// TIA Portal V18 export
FUNCTION "SS2_A4_32DO_IO_Update" : Void   // FC11150, LAD
{ S7_Optimized_Access := 'TRUE' }
VERSION : 0.1
// stored: AutoNumber false, IsIECCheckEnabled false, SetENOAutomatically false, UDAEnableTagReadback false
BEGIN

REGION Network 1: DQa0
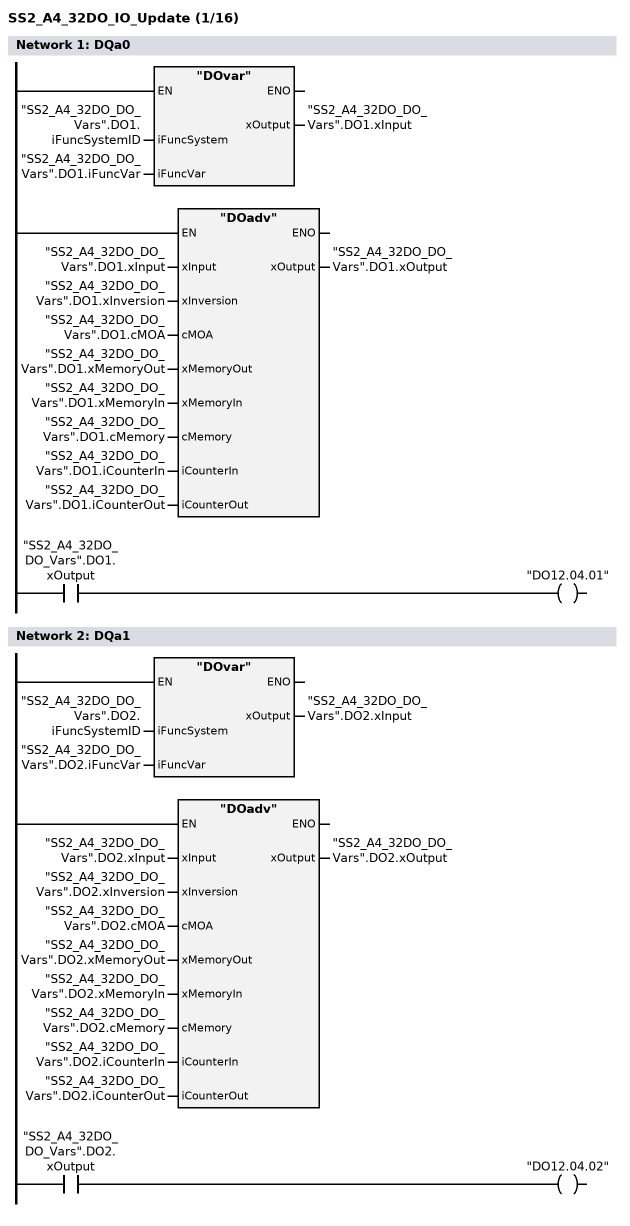
   RUNG wire#powerrail
      "DOvar"(iFuncSystem := "SS2_A4_32DO_DO_Vars".DO1.iFuncSystemID, iFuncVar := "SS2_A4_32DO_DO_Vars".DO1.iFuncVar, xOutput => "SS2_A4_32DO_DO_Vars".DO1.xInput)
   END_RUNG
   RUNG wire#powerrail
      "DOadv"(xInput := "SS2_A4_32DO_DO_Vars".DO1.xInput, xInversion := "SS2_A4_32DO_DO_Vars".DO1.xInversion, cMOA := "SS2_A4_32DO_DO_Vars".DO1.cMOA, xMemoryOut := "SS2_A4_32DO_DO_Vars".DO1.xMemoryOut, xMemoryIn := "SS2_A4_32DO_DO_Vars".DO1.xMemoryIn, cMemory := "SS2_A4_32DO_DO_Vars".DO1.cMemory, iCounterIn := "SS2_A4_32DO_DO_Vars".DO1.iCounterIn, iCounterOut := "SS2_A4_32DO_DO_Vars".DO1.iCounterOut, xOutput => "SS2_A4_32DO_DO_Vars".DO1.xOutput)
   END_RUNG
   RUNG wire#powerrail
      Contact( "SS2_A4_32DO_DO_Vars".DO1.xOutput )
      Coil( "DO12.04.01" )
   END_RUNG
   // the same network as SCL:
   "DOvar"(iFuncSystem := "SS2_A4_32DO_DO_Vars".DO1.iFuncSystemID,
           iFuncVar := "SS2_A4_32DO_DO_Vars".DO1.iFuncVar,
           xOutput => "SS2_A4_32DO_DO_Vars".DO1.xInput);
   "DOadv"(xInput := "SS2_A4_32DO_DO_Vars".DO1.xInput,
           xInversion := "SS2_A4_32DO_DO_Vars".DO1.xInversion,
           cMOA := "SS2_A4_32DO_DO_Vars".DO1.cMOA,
           xMemoryOut := "SS2_A4_32DO_DO_Vars".DO1.xMemoryOut,
           xMemoryIn := "SS2_A4_32DO_DO_Vars".DO1.xMemoryIn,
           cMemory := "SS2_A4_32DO_DO_Vars".DO1.cMemory,
           iCounterIn := "SS2_A4_32DO_DO_Vars".DO1.iCounterIn,
           iCounterOut := "SS2_A4_32DO_DO_Vars".DO1.iCounterOut,
           xOutput => "SS2_A4_32DO_DO_Vars".DO1.xOutput);
   "DO12.04.01" := "SS2_A4_32DO_DO_Vars".DO1.xOutput;
END_REGION

REGION Network 2: DQa1
   RUNG wire#powerrail
      "DOvar"(iFuncSystem := "SS2_A4_32DO_DO_Vars".DO2.iFuncSystemID, iFuncVar := "SS2_A4_32DO_DO_Vars".DO2.iFuncVar, xOutput => "SS2_A4_32DO_DO_Vars".DO2.xInput)
   END_RUNG
   RUNG wire#powerrail
      "DOadv"(xInput := "SS2_A4_32DO_DO_Vars".DO2.xInput, xInversion := "SS2_A4_32DO_DO_Vars".DO2.xInversion, cMOA := "SS2_A4_32DO_DO_Vars".DO2.cMOA, xMemoryOut := "SS2_A4_32DO_DO_Vars".DO2.xMemoryOut, xMemoryIn := "SS2_A4_32DO_DO_Vars".DO2.xMemoryIn, cMemory := "SS2_A4_32DO_DO_Vars".DO2.cMemory, iCounterIn := "SS2_A4_32DO_DO_Vars".DO2.iCounterIn, iCounterOut := "SS2_A4_32DO_DO_Vars".DO2.iCounterOut, xOutput => "SS2_A4_32DO_DO_Vars".DO2.xOutput)
   END_RUNG
   RUNG wire#powerrail
      Contact( "SS2_A4_32DO_DO_Vars".DO2.xOutput )
      Coil( "DO12.04.02" )
   END_RUNG
   // the same network as SCL:
   "DOvar"(iFuncSystem := "SS2_A4_32DO_DO_Vars".DO2.iFuncSystemID,
           iFuncVar := "SS2_A4_32DO_DO_Vars".DO2.iFuncVar,
           xOutput => "SS2_A4_32DO_DO_Vars".DO2.xInput);
   "DOadv"(xInput := "SS2_A4_32DO_DO_Vars".DO2.xInput,
           xInversion := "SS2_A4_32DO_DO_Vars".DO2.xInversion,
           cMOA := "SS2_A4_32DO_DO_Vars".DO2.cMOA,
           xMemoryOut := "SS2_A4_32DO_DO_Vars".DO2.xMemoryOut,
           xMemoryIn := "SS2_A4_32DO_DO_Vars".DO2.xMemoryIn,
           cMemory := "SS2_A4_32DO_DO_Vars".DO2.cMemory,
           iCounterIn := "SS2_A4_32DO_DO_Vars".DO2.iCounterIn,
           iCounterOut := "SS2_A4_32DO_DO_Vars".DO2.iCounterOut,
           xOutput => "SS2_A4_32DO_DO_Vars".DO2.xOutput);
   "DO12.04.02" := "SS2_A4_32DO_DO_Vars".DO2.xOutput;
END_REGION

REGION Network 3: DQa2
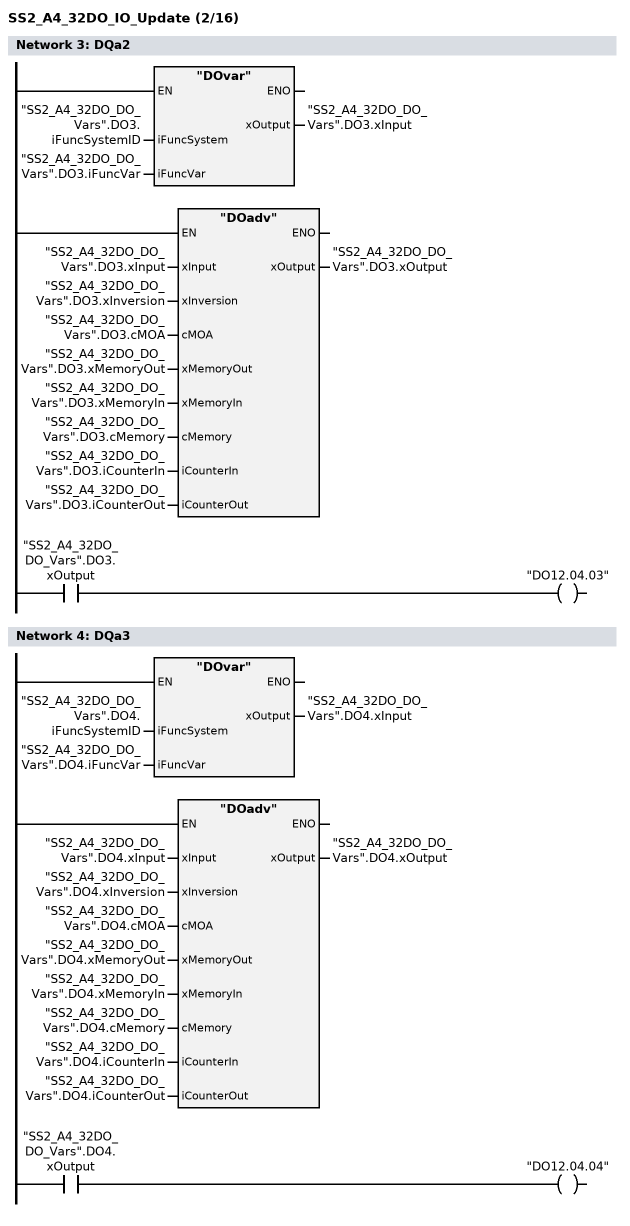
   RUNG wire#powerrail
      "DOvar"(iFuncSystem := "SS2_A4_32DO_DO_Vars".DO3.iFuncSystemID, iFuncVar := "SS2_A4_32DO_DO_Vars".DO3.iFuncVar, xOutput => "SS2_A4_32DO_DO_Vars".DO3.xInput)
   END_RUNG
   RUNG wire#powerrail
      "DOadv"(xInput := "SS2_A4_32DO_DO_Vars".DO3.xInput, xInversion := "SS2_A4_32DO_DO_Vars".DO3.xInversion, cMOA := "SS2_A4_32DO_DO_Vars".DO3.cMOA, xMemoryOut := "SS2_A4_32DO_DO_Vars".DO3.xMemoryOut, xMemoryIn := "SS2_A4_32DO_DO_Vars".DO3.xMemoryIn, cMemory := "SS2_A4_32DO_DO_Vars".DO3.cMemory, iCounterIn := "SS2_A4_32DO_DO_Vars".DO3.iCounterIn, iCounterOut := "SS2_A4_32DO_DO_Vars".DO3.iCounterOut, xOutput => "SS2_A4_32DO_DO_Vars".DO3.xOutput)
   END_RUNG
   RUNG wire#powerrail
      Contact( "SS2_A4_32DO_DO_Vars".DO3.xOutput )
      Coil( "DO12.04.03" )
   END_RUNG
   // the same network as SCL:
   "DOvar"(iFuncSystem := "SS2_A4_32DO_DO_Vars".DO3.iFuncSystemID,
           iFuncVar := "SS2_A4_32DO_DO_Vars".DO3.iFuncVar,
           xOutput => "SS2_A4_32DO_DO_Vars".DO3.xInput);
   "DOadv"(xInput := "SS2_A4_32DO_DO_Vars".DO3.xInput,
           xInversion := "SS2_A4_32DO_DO_Vars".DO3.xInversion,
           cMOA := "SS2_A4_32DO_DO_Vars".DO3.cMOA,
           xMemoryOut := "SS2_A4_32DO_DO_Vars".DO3.xMemoryOut,
           xMemoryIn := "SS2_A4_32DO_DO_Vars".DO3.xMemoryIn,
           cMemory := "SS2_A4_32DO_DO_Vars".DO3.cMemory,
           iCounterIn := "SS2_A4_32DO_DO_Vars".DO3.iCounterIn,
           iCounterOut := "SS2_A4_32DO_DO_Vars".DO3.iCounterOut,
           xOutput => "SS2_A4_32DO_DO_Vars".DO3.xOutput);
   "DO12.04.03" := "SS2_A4_32DO_DO_Vars".DO3.xOutput;
END_REGION

REGION Network 4: DQa3
   RUNG wire#powerrail
      "DOvar"(iFuncSystem := "SS2_A4_32DO_DO_Vars".DO4.iFuncSystemID, iFuncVar := "SS2_A4_32DO_DO_Vars".DO4.iFuncVar, xOutput => "SS2_A4_32DO_DO_Vars".DO4.xInput)
   END_RUNG
   RUNG wire#powerrail
      "DOadv"(xInput := "SS2_A4_32DO_DO_Vars".DO4.xInput, xInversion := "SS2_A4_32DO_DO_Vars".DO4.xInversion, cMOA := "SS2_A4_32DO_DO_Vars".DO4.cMOA, xMemoryOut := "SS2_A4_32DO_DO_Vars".DO4.xMemoryOut, xMemoryIn := "SS2_A4_32DO_DO_Vars".DO4.xMemoryIn, cMemory := "SS2_A4_32DO_DO_Vars".DO4.cMemory, iCounterIn := "SS2_A4_32DO_DO_Vars".DO4.iCounterIn, iCounterOut := "SS2_A4_32DO_DO_Vars".DO4.iCounterOut, xOutput => "SS2_A4_32DO_DO_Vars".DO4.xOutput)
   END_RUNG
   RUNG wire#powerrail
      Contact( "SS2_A4_32DO_DO_Vars".DO4.xOutput )
      Coil( "DO12.04.04" )
   END_RUNG
   // the same network as SCL:
   "DOvar"(iFuncSystem := "SS2_A4_32DO_DO_Vars".DO4.iFuncSystemID,
           iFuncVar := "SS2_A4_32DO_DO_Vars".DO4.iFuncVar,
           xOutput => "SS2_A4_32DO_DO_Vars".DO4.xInput);
   "DOadv"(xInput := "SS2_A4_32DO_DO_Vars".DO4.xInput,
           xInversion := "SS2_A4_32DO_DO_Vars".DO4.xInversion,
           cMOA := "SS2_A4_32DO_DO_Vars".DO4.cMOA,
           xMemoryOut := "SS2_A4_32DO_DO_Vars".DO4.xMemoryOut,
           xMemoryIn := "SS2_A4_32DO_DO_Vars".DO4.xMemoryIn,
           cMemory := "SS2_A4_32DO_DO_Vars".DO4.cMemory,
           iCounterIn := "SS2_A4_32DO_DO_Vars".DO4.iCounterIn,
           iCounterOut := "SS2_A4_32DO_DO_Vars".DO4.iCounterOut,
           xOutput => "SS2_A4_32DO_DO_Vars".DO4.xOutput);
   "DO12.04.04" := "SS2_A4_32DO_DO_Vars".DO4.xOutput;
END_REGION

REGION Network 5: DQa4
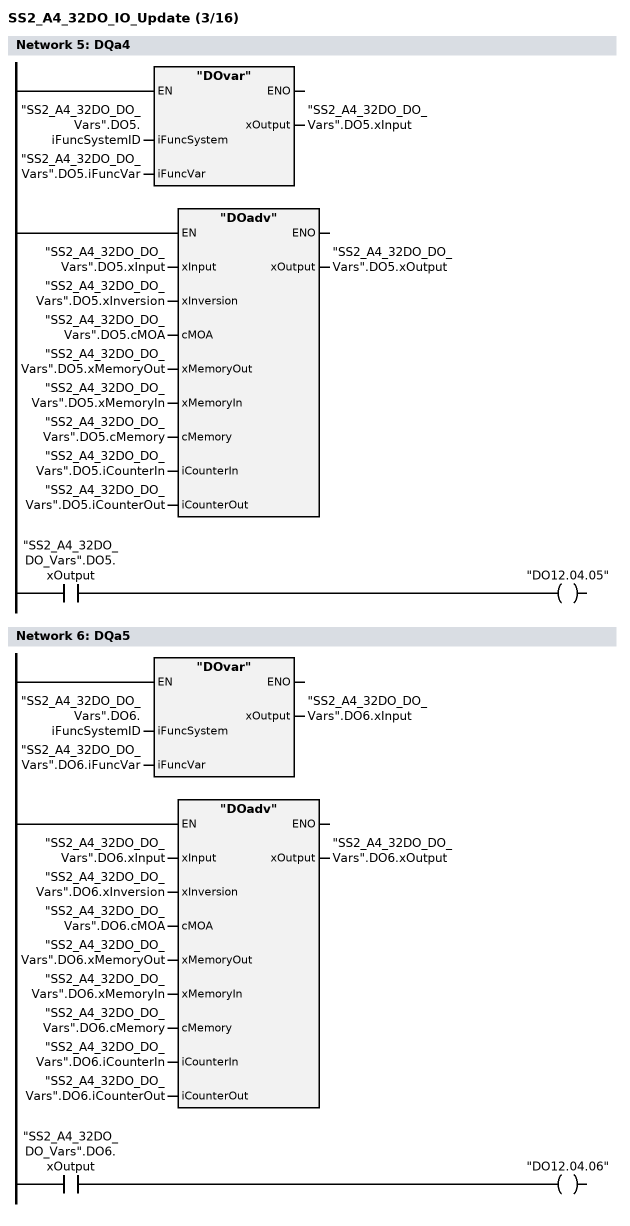
   RUNG wire#powerrail
      "DOvar"(iFuncSystem := "SS2_A4_32DO_DO_Vars".DO5.iFuncSystemID, iFuncVar := "SS2_A4_32DO_DO_Vars".DO5.iFuncVar, xOutput => "SS2_A4_32DO_DO_Vars".DO5.xInput)
   END_RUNG
   RUNG wire#powerrail
      "DOadv"(xInput := "SS2_A4_32DO_DO_Vars".DO5.xInput, xInversion := "SS2_A4_32DO_DO_Vars".DO5.xInversion, cMOA := "SS2_A4_32DO_DO_Vars".DO5.cMOA, xMemoryOut := "SS2_A4_32DO_DO_Vars".DO5.xMemoryOut, xMemoryIn := "SS2_A4_32DO_DO_Vars".DO5.xMemoryIn, cMemory := "SS2_A4_32DO_DO_Vars".DO5.cMemory, iCounterIn := "SS2_A4_32DO_DO_Vars".DO5.iCounterIn, iCounterOut := "SS2_A4_32DO_DO_Vars".DO5.iCounterOut, xOutput => "SS2_A4_32DO_DO_Vars".DO5.xOutput)
   END_RUNG
   RUNG wire#powerrail
      Contact( "SS2_A4_32DO_DO_Vars".DO5.xOutput )
      Coil( "DO12.04.05" )
   END_RUNG
   // the same network as SCL:
   "DOvar"(iFuncSystem := "SS2_A4_32DO_DO_Vars".DO5.iFuncSystemID,
           iFuncVar := "SS2_A4_32DO_DO_Vars".DO5.iFuncVar,
           xOutput => "SS2_A4_32DO_DO_Vars".DO5.xInput);
   "DOadv"(xInput := "SS2_A4_32DO_DO_Vars".DO5.xInput,
           xInversion := "SS2_A4_32DO_DO_Vars".DO5.xInversion,
           cMOA := "SS2_A4_32DO_DO_Vars".DO5.cMOA,
           xMemoryOut := "SS2_A4_32DO_DO_Vars".DO5.xMemoryOut,
           xMemoryIn := "SS2_A4_32DO_DO_Vars".DO5.xMemoryIn,
           cMemory := "SS2_A4_32DO_DO_Vars".DO5.cMemory,
           iCounterIn := "SS2_A4_32DO_DO_Vars".DO5.iCounterIn,
           iCounterOut := "SS2_A4_32DO_DO_Vars".DO5.iCounterOut,
           xOutput => "SS2_A4_32DO_DO_Vars".DO5.xOutput);
   "DO12.04.05" := "SS2_A4_32DO_DO_Vars".DO5.xOutput;
END_REGION

REGION Network 6: DQa5
   RUNG wire#powerrail
      "DOvar"(iFuncSystem := "SS2_A4_32DO_DO_Vars".DO6.iFuncSystemID, iFuncVar := "SS2_A4_32DO_DO_Vars".DO6.iFuncVar, xOutput => "SS2_A4_32DO_DO_Vars".DO6.xInput)
   END_RUNG
   RUNG wire#powerrail
      "DOadv"(xInput := "SS2_A4_32DO_DO_Vars".DO6.xInput, xInversion := "SS2_A4_32DO_DO_Vars".DO6.xInversion, cMOA := "SS2_A4_32DO_DO_Vars".DO6.cMOA, xMemoryOut := "SS2_A4_32DO_DO_Vars".DO6.xMemoryOut, xMemoryIn := "SS2_A4_32DO_DO_Vars".DO6.xMemoryIn, cMemory := "SS2_A4_32DO_DO_Vars".DO6.cMemory, iCounterIn := "SS2_A4_32DO_DO_Vars".DO6.iCounterIn, iCounterOut := "SS2_A4_32DO_DO_Vars".DO6.iCounterOut, xOutput => "SS2_A4_32DO_DO_Vars".DO6.xOutput)
   END_RUNG
   RUNG wire#powerrail
      Contact( "SS2_A4_32DO_DO_Vars".DO6.xOutput )
      Coil( "DO12.04.06" )
   END_RUNG
   // the same network as SCL:
   "DOvar"(iFuncSystem := "SS2_A4_32DO_DO_Vars".DO6.iFuncSystemID,
           iFuncVar := "SS2_A4_32DO_DO_Vars".DO6.iFuncVar,
           xOutput => "SS2_A4_32DO_DO_Vars".DO6.xInput);
   "DOadv"(xInput := "SS2_A4_32DO_DO_Vars".DO6.xInput,
           xInversion := "SS2_A4_32DO_DO_Vars".DO6.xInversion,
           cMOA := "SS2_A4_32DO_DO_Vars".DO6.cMOA,
           xMemoryOut := "SS2_A4_32DO_DO_Vars".DO6.xMemoryOut,
           xMemoryIn := "SS2_A4_32DO_DO_Vars".DO6.xMemoryIn,
           cMemory := "SS2_A4_32DO_DO_Vars".DO6.cMemory,
           iCounterIn := "SS2_A4_32DO_DO_Vars".DO6.iCounterIn,
           iCounterOut := "SS2_A4_32DO_DO_Vars".DO6.iCounterOut,
           xOutput => "SS2_A4_32DO_DO_Vars".DO6.xOutput);
   "DO12.04.06" := "SS2_A4_32DO_DO_Vars".DO6.xOutput;
END_REGION

REGION Network 7: DQa6
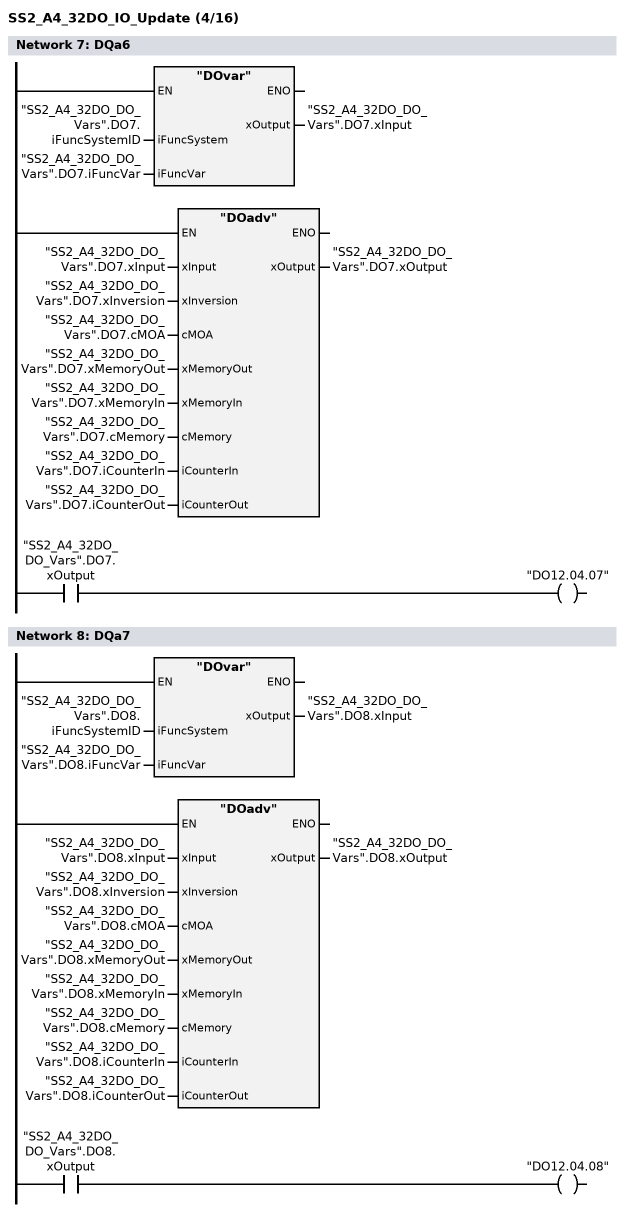
   RUNG wire#powerrail
      "DOvar"(iFuncSystem := "SS2_A4_32DO_DO_Vars".DO7.iFuncSystemID, iFuncVar := "SS2_A4_32DO_DO_Vars".DO7.iFuncVar, xOutput => "SS2_A4_32DO_DO_Vars".DO7.xInput)
   END_RUNG
   RUNG wire#powerrail
      "DOadv"(xInput := "SS2_A4_32DO_DO_Vars".DO7.xInput, xInversion := "SS2_A4_32DO_DO_Vars".DO7.xInversion, cMOA := "SS2_A4_32DO_DO_Vars".DO7.cMOA, xMemoryOut := "SS2_A4_32DO_DO_Vars".DO7.xMemoryOut, xMemoryIn := "SS2_A4_32DO_DO_Vars".DO7.xMemoryIn, cMemory := "SS2_A4_32DO_DO_Vars".DO7.cMemory, iCounterIn := "SS2_A4_32DO_DO_Vars".DO7.iCounterIn, iCounterOut := "SS2_A4_32DO_DO_Vars".DO7.iCounterOut, xOutput => "SS2_A4_32DO_DO_Vars".DO7.xOutput)
   END_RUNG
   RUNG wire#powerrail
      Contact( "SS2_A4_32DO_DO_Vars".DO7.xOutput )
      Coil( "DO12.04.07" )
   END_RUNG
   // the same network as SCL:
   "DOvar"(iFuncSystem := "SS2_A4_32DO_DO_Vars".DO7.iFuncSystemID,
           iFuncVar := "SS2_A4_32DO_DO_Vars".DO7.iFuncVar,
           xOutput => "SS2_A4_32DO_DO_Vars".DO7.xInput);
   "DOadv"(xInput := "SS2_A4_32DO_DO_Vars".DO7.xInput,
           xInversion := "SS2_A4_32DO_DO_Vars".DO7.xInversion,
           cMOA := "SS2_A4_32DO_DO_Vars".DO7.cMOA,
           xMemoryOut := "SS2_A4_32DO_DO_Vars".DO7.xMemoryOut,
           xMemoryIn := "SS2_A4_32DO_DO_Vars".DO7.xMemoryIn,
           cMemory := "SS2_A4_32DO_DO_Vars".DO7.cMemory,
           iCounterIn := "SS2_A4_32DO_DO_Vars".DO7.iCounterIn,
           iCounterOut := "SS2_A4_32DO_DO_Vars".DO7.iCounterOut,
           xOutput => "SS2_A4_32DO_DO_Vars".DO7.xOutput);
   "DO12.04.07" := "SS2_A4_32DO_DO_Vars".DO7.xOutput;
END_REGION

REGION Network 8: DQa7
   RUNG wire#powerrail
      "DOvar"(iFuncSystem := "SS2_A4_32DO_DO_Vars".DO8.iFuncSystemID, iFuncVar := "SS2_A4_32DO_DO_Vars".DO8.iFuncVar, xOutput => "SS2_A4_32DO_DO_Vars".DO8.xInput)
   END_RUNG
   RUNG wire#powerrail
      "DOadv"(xInput := "SS2_A4_32DO_DO_Vars".DO8.xInput, xInversion := "SS2_A4_32DO_DO_Vars".DO8.xInversion, cMOA := "SS2_A4_32DO_DO_Vars".DO8.cMOA, xMemoryOut := "SS2_A4_32DO_DO_Vars".DO8.xMemoryOut, xMemoryIn := "SS2_A4_32DO_DO_Vars".DO8.xMemoryIn, cMemory := "SS2_A4_32DO_DO_Vars".DO8.cMemory, iCounterIn := "SS2_A4_32DO_DO_Vars".DO8.iCounterIn, iCounterOut := "SS2_A4_32DO_DO_Vars".DO8.iCounterOut, xOutput => "SS2_A4_32DO_DO_Vars".DO8.xOutput)
   END_RUNG
   RUNG wire#powerrail
      Contact( "SS2_A4_32DO_DO_Vars".DO8.xOutput )
      Coil( "DO12.04.08" )
   END_RUNG
   // the same network as SCL:
   "DOvar"(iFuncSystem := "SS2_A4_32DO_DO_Vars".DO8.iFuncSystemID,
           iFuncVar := "SS2_A4_32DO_DO_Vars".DO8.iFuncVar,
           xOutput => "SS2_A4_32DO_DO_Vars".DO8.xInput);
   "DOadv"(xInput := "SS2_A4_32DO_DO_Vars".DO8.xInput,
           xInversion := "SS2_A4_32DO_DO_Vars".DO8.xInversion,
           cMOA := "SS2_A4_32DO_DO_Vars".DO8.cMOA,
           xMemoryOut := "SS2_A4_32DO_DO_Vars".DO8.xMemoryOut,
           xMemoryIn := "SS2_A4_32DO_DO_Vars".DO8.xMemoryIn,
           cMemory := "SS2_A4_32DO_DO_Vars".DO8.cMemory,
           iCounterIn := "SS2_A4_32DO_DO_Vars".DO8.iCounterIn,
           iCounterOut := "SS2_A4_32DO_DO_Vars".DO8.iCounterOut,
           xOutput => "SS2_A4_32DO_DO_Vars".DO8.xOutput);
   "DO12.04.08" := "SS2_A4_32DO_DO_Vars".DO8.xOutput;
END_REGION

REGION Network 9: DQb0
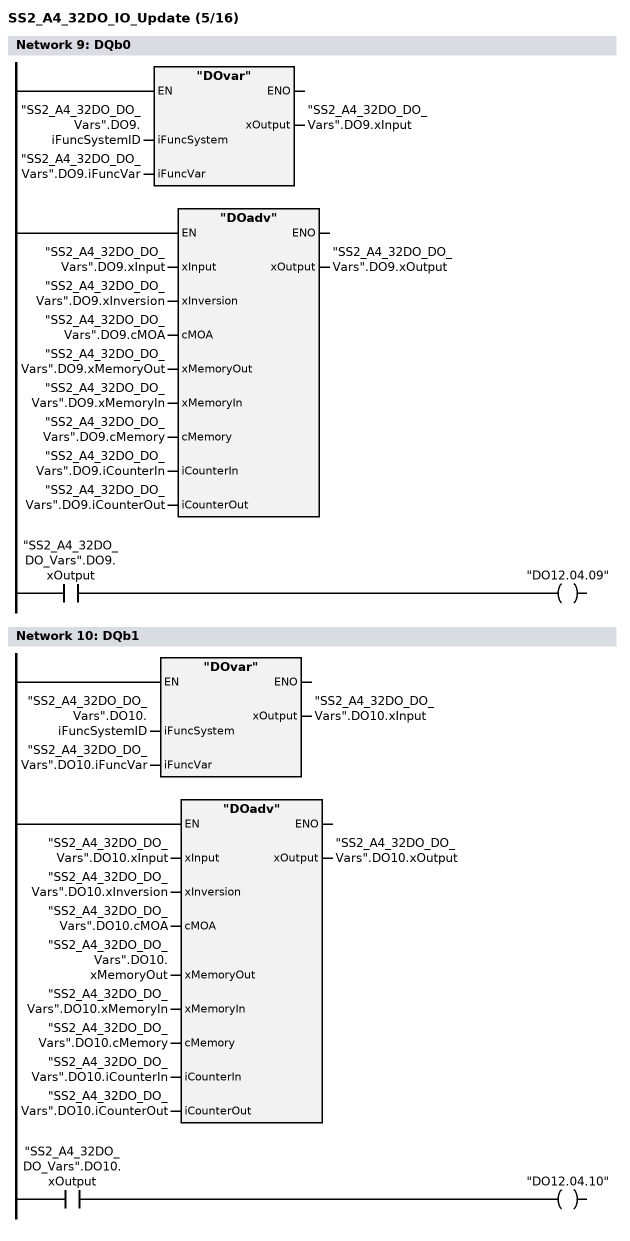
   RUNG wire#powerrail
      "DOvar"(iFuncSystem := "SS2_A4_32DO_DO_Vars".DO9.iFuncSystemID, iFuncVar := "SS2_A4_32DO_DO_Vars".DO9.iFuncVar, xOutput => "SS2_A4_32DO_DO_Vars".DO9.xInput)
   END_RUNG
   RUNG wire#powerrail
      "DOadv"(xInput := "SS2_A4_32DO_DO_Vars".DO9.xInput, xInversion := "SS2_A4_32DO_DO_Vars".DO9.xInversion, cMOA := "SS2_A4_32DO_DO_Vars".DO9.cMOA, xMemoryOut := "SS2_A4_32DO_DO_Vars".DO9.xMemoryOut, xMemoryIn := "SS2_A4_32DO_DO_Vars".DO9.xMemoryIn, cMemory := "SS2_A4_32DO_DO_Vars".DO9.cMemory, iCounterIn := "SS2_A4_32DO_DO_Vars".DO9.iCounterIn, iCounterOut := "SS2_A4_32DO_DO_Vars".DO9.iCounterOut, xOutput => "SS2_A4_32DO_DO_Vars".DO9.xOutput)
   END_RUNG
   RUNG wire#powerrail
      Contact( "SS2_A4_32DO_DO_Vars".DO9.xOutput )
      Coil( "DO12.04.09" )
   END_RUNG
   // the same network as SCL:
   "DOvar"(iFuncSystem := "SS2_A4_32DO_DO_Vars".DO9.iFuncSystemID,
           iFuncVar := "SS2_A4_32DO_DO_Vars".DO9.iFuncVar,
           xOutput => "SS2_A4_32DO_DO_Vars".DO9.xInput);
   "DOadv"(xInput := "SS2_A4_32DO_DO_Vars".DO9.xInput,
           xInversion := "SS2_A4_32DO_DO_Vars".DO9.xInversion,
           cMOA := "SS2_A4_32DO_DO_Vars".DO9.cMOA,
           xMemoryOut := "SS2_A4_32DO_DO_Vars".DO9.xMemoryOut,
           xMemoryIn := "SS2_A4_32DO_DO_Vars".DO9.xMemoryIn,
           cMemory := "SS2_A4_32DO_DO_Vars".DO9.cMemory,
           iCounterIn := "SS2_A4_32DO_DO_Vars".DO9.iCounterIn,
           iCounterOut := "SS2_A4_32DO_DO_Vars".DO9.iCounterOut,
           xOutput => "SS2_A4_32DO_DO_Vars".DO9.xOutput);
   "DO12.04.09" := "SS2_A4_32DO_DO_Vars".DO9.xOutput;
END_REGION

REGION Network 10: DQb1
   RUNG wire#powerrail
      "DOvar"(iFuncSystem := "SS2_A4_32DO_DO_Vars".DO10.iFuncSystemID, iFuncVar := "SS2_A4_32DO_DO_Vars".DO10.iFuncVar, xOutput => "SS2_A4_32DO_DO_Vars".DO10.xInput)
   END_RUNG
   RUNG wire#powerrail
      "DOadv"(xInput := "SS2_A4_32DO_DO_Vars".DO10.xInput, xInversion := "SS2_A4_32DO_DO_Vars".DO10.xInversion, cMOA := "SS2_A4_32DO_DO_Vars".DO10.cMOA, xMemoryOut := "SS2_A4_32DO_DO_Vars".DO10.xMemoryOut, xMemoryIn := "SS2_A4_32DO_DO_Vars".DO10.xMemoryIn, cMemory := "SS2_A4_32DO_DO_Vars".DO10.cMemory, iCounterIn := "SS2_A4_32DO_DO_Vars".DO10.iCounterIn, iCounterOut := "SS2_A4_32DO_DO_Vars".DO10.iCounterOut, xOutput => "SS2_A4_32DO_DO_Vars".DO10.xOutput)
   END_RUNG
   RUNG wire#powerrail
      Contact( "SS2_A4_32DO_DO_Vars".DO10.xOutput )
      Coil( "DO12.04.10" )
   END_RUNG
   // the same network as SCL:
   "DOvar"(iFuncSystem := "SS2_A4_32DO_DO_Vars".DO10.iFuncSystemID,
           iFuncVar := "SS2_A4_32DO_DO_Vars".DO10.iFuncVar,
           xOutput => "SS2_A4_32DO_DO_Vars".DO10.xInput);
   "DOadv"(xInput := "SS2_A4_32DO_DO_Vars".DO10.xInput,
           xInversion := "SS2_A4_32DO_DO_Vars".DO10.xInversion,
           cMOA := "SS2_A4_32DO_DO_Vars".DO10.cMOA,
           xMemoryOut := "SS2_A4_32DO_DO_Vars".DO10.xMemoryOut,
           xMemoryIn := "SS2_A4_32DO_DO_Vars".DO10.xMemoryIn,
           cMemory := "SS2_A4_32DO_DO_Vars".DO10.cMemory,
           iCounterIn := "SS2_A4_32DO_DO_Vars".DO10.iCounterIn,
           iCounterOut := "SS2_A4_32DO_DO_Vars".DO10.iCounterOut,
           xOutput => "SS2_A4_32DO_DO_Vars".DO10.xOutput);
   "DO12.04.10" := "SS2_A4_32DO_DO_Vars".DO10.xOutput;
END_REGION

REGION Network 11: DQb2
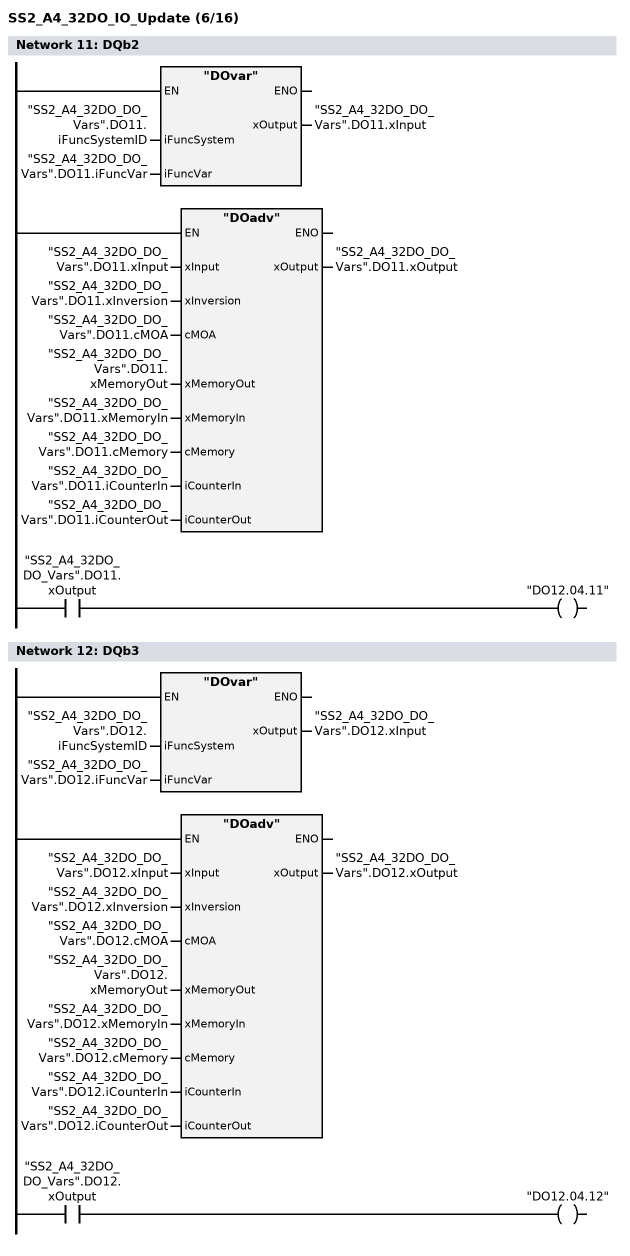
   RUNG wire#powerrail
      "DOvar"(iFuncSystem := "SS2_A4_32DO_DO_Vars".DO11.iFuncSystemID, iFuncVar := "SS2_A4_32DO_DO_Vars".DO11.iFuncVar, xOutput => "SS2_A4_32DO_DO_Vars".DO11.xInput)
   END_RUNG
   RUNG wire#powerrail
      "DOadv"(xInput := "SS2_A4_32DO_DO_Vars".DO11.xInput, xInversion := "SS2_A4_32DO_DO_Vars".DO11.xInversion, cMOA := "SS2_A4_32DO_DO_Vars".DO11.cMOA, xMemoryOut := "SS2_A4_32DO_DO_Vars".DO11.xMemoryOut, xMemoryIn := "SS2_A4_32DO_DO_Vars".DO11.xMemoryIn, cMemory := "SS2_A4_32DO_DO_Vars".DO11.cMemory, iCounterIn := "SS2_A4_32DO_DO_Vars".DO11.iCounterIn, iCounterOut := "SS2_A4_32DO_DO_Vars".DO11.iCounterOut, xOutput => "SS2_A4_32DO_DO_Vars".DO11.xOutput)
   END_RUNG
   RUNG wire#powerrail
      Contact( "SS2_A4_32DO_DO_Vars".DO11.xOutput )
      Coil( "DO12.04.11" )
   END_RUNG
   // the same network as SCL:
   "DOvar"(iFuncSystem := "SS2_A4_32DO_DO_Vars".DO11.iFuncSystemID,
           iFuncVar := "SS2_A4_32DO_DO_Vars".DO11.iFuncVar,
           xOutput => "SS2_A4_32DO_DO_Vars".DO11.xInput);
   "DOadv"(xInput := "SS2_A4_32DO_DO_Vars".DO11.xInput,
           xInversion := "SS2_A4_32DO_DO_Vars".DO11.xInversion,
           cMOA := "SS2_A4_32DO_DO_Vars".DO11.cMOA,
           xMemoryOut := "SS2_A4_32DO_DO_Vars".DO11.xMemoryOut,
           xMemoryIn := "SS2_A4_32DO_DO_Vars".DO11.xMemoryIn,
           cMemory := "SS2_A4_32DO_DO_Vars".DO11.cMemory,
           iCounterIn := "SS2_A4_32DO_DO_Vars".DO11.iCounterIn,
           iCounterOut := "SS2_A4_32DO_DO_Vars".DO11.iCounterOut,
           xOutput => "SS2_A4_32DO_DO_Vars".DO11.xOutput);
   "DO12.04.11" := "SS2_A4_32DO_DO_Vars".DO11.xOutput;
END_REGION

REGION Network 12: DQb3
   RUNG wire#powerrail
      "DOvar"(iFuncSystem := "SS2_A4_32DO_DO_Vars".DO12.iFuncSystemID, iFuncVar := "SS2_A4_32DO_DO_Vars".DO12.iFuncVar, xOutput => "SS2_A4_32DO_DO_Vars".DO12.xInput)
   END_RUNG
   RUNG wire#powerrail
      "DOadv"(xInput := "SS2_A4_32DO_DO_Vars".DO12.xInput, xInversion := "SS2_A4_32DO_DO_Vars".DO12.xInversion, cMOA := "SS2_A4_32DO_DO_Vars".DO12.cMOA, xMemoryOut := "SS2_A4_32DO_DO_Vars".DO12.xMemoryOut, xMemoryIn := "SS2_A4_32DO_DO_Vars".DO12.xMemoryIn, cMemory := "SS2_A4_32DO_DO_Vars".DO12.cMemory, iCounterIn := "SS2_A4_32DO_DO_Vars".DO12.iCounterIn, iCounterOut := "SS2_A4_32DO_DO_Vars".DO12.iCounterOut, xOutput => "SS2_A4_32DO_DO_Vars".DO12.xOutput)
   END_RUNG
   RUNG wire#powerrail
      Contact( "SS2_A4_32DO_DO_Vars".DO12.xOutput )
      Coil( "DO12.04.12" )
   END_RUNG
   // the same network as SCL:
   "DOvar"(iFuncSystem := "SS2_A4_32DO_DO_Vars".DO12.iFuncSystemID,
           iFuncVar := "SS2_A4_32DO_DO_Vars".DO12.iFuncVar,
           xOutput => "SS2_A4_32DO_DO_Vars".DO12.xInput);
   "DOadv"(xInput := "SS2_A4_32DO_DO_Vars".DO12.xInput,
           xInversion := "SS2_A4_32DO_DO_Vars".DO12.xInversion,
           cMOA := "SS2_A4_32DO_DO_Vars".DO12.cMOA,
           xMemoryOut := "SS2_A4_32DO_DO_Vars".DO12.xMemoryOut,
           xMemoryIn := "SS2_A4_32DO_DO_Vars".DO12.xMemoryIn,
           cMemory := "SS2_A4_32DO_DO_Vars".DO12.cMemory,
           iCounterIn := "SS2_A4_32DO_DO_Vars".DO12.iCounterIn,
           iCounterOut := "SS2_A4_32DO_DO_Vars".DO12.iCounterOut,
           xOutput => "SS2_A4_32DO_DO_Vars".DO12.xOutput);
   "DO12.04.12" := "SS2_A4_32DO_DO_Vars".DO12.xOutput;
END_REGION

REGION Network 13: DQb4
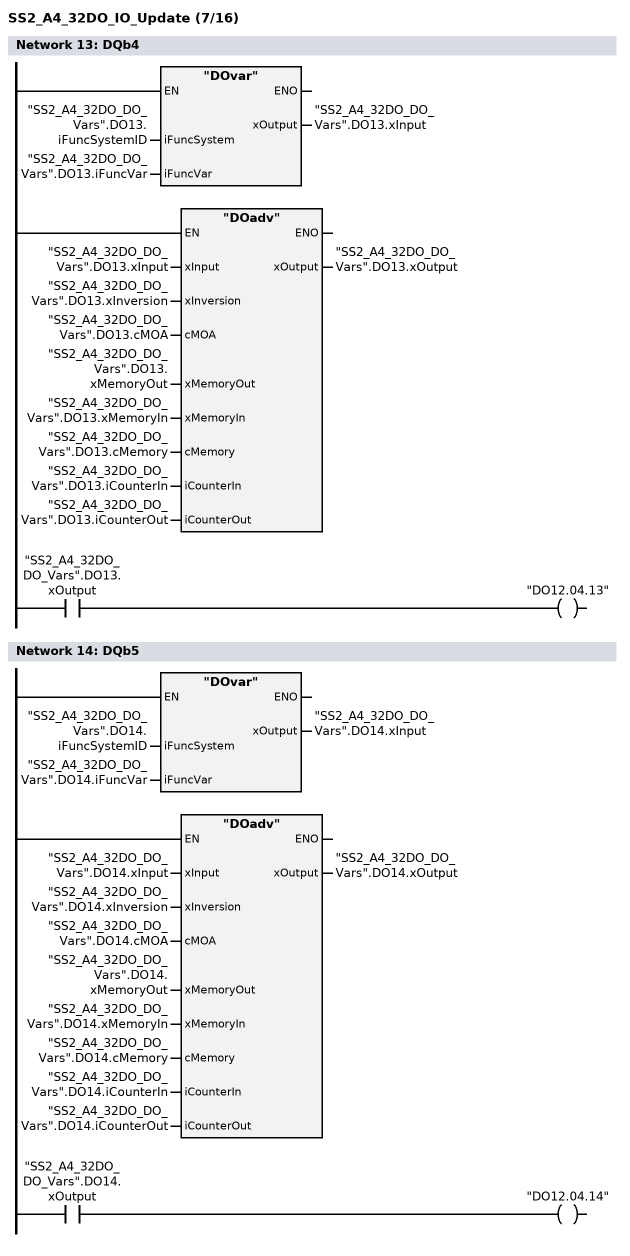
   RUNG wire#powerrail
      "DOvar"(iFuncSystem := "SS2_A4_32DO_DO_Vars".DO13.iFuncSystemID, iFuncVar := "SS2_A4_32DO_DO_Vars".DO13.iFuncVar, xOutput => "SS2_A4_32DO_DO_Vars".DO13.xInput)
   END_RUNG
   RUNG wire#powerrail
      "DOadv"(xInput := "SS2_A4_32DO_DO_Vars".DO13.xInput, xInversion := "SS2_A4_32DO_DO_Vars".DO13.xInversion, cMOA := "SS2_A4_32DO_DO_Vars".DO13.cMOA, xMemoryOut := "SS2_A4_32DO_DO_Vars".DO13.xMemoryOut, xMemoryIn := "SS2_A4_32DO_DO_Vars".DO13.xMemoryIn, cMemory := "SS2_A4_32DO_DO_Vars".DO13.cMemory, iCounterIn := "SS2_A4_32DO_DO_Vars".DO13.iCounterIn, iCounterOut := "SS2_A4_32DO_DO_Vars".DO13.iCounterOut, xOutput => "SS2_A4_32DO_DO_Vars".DO13.xOutput)
   END_RUNG
   RUNG wire#powerrail
      Contact( "SS2_A4_32DO_DO_Vars".DO13.xOutput )
      Coil( "DO12.04.13" )
   END_RUNG
   // the same network as SCL:
   "DOvar"(iFuncSystem := "SS2_A4_32DO_DO_Vars".DO13.iFuncSystemID,
           iFuncVar := "SS2_A4_32DO_DO_Vars".DO13.iFuncVar,
           xOutput => "SS2_A4_32DO_DO_Vars".DO13.xInput);
   "DOadv"(xInput := "SS2_A4_32DO_DO_Vars".DO13.xInput,
           xInversion := "SS2_A4_32DO_DO_Vars".DO13.xInversion,
           cMOA := "SS2_A4_32DO_DO_Vars".DO13.cMOA,
           xMemoryOut := "SS2_A4_32DO_DO_Vars".DO13.xMemoryOut,
           xMemoryIn := "SS2_A4_32DO_DO_Vars".DO13.xMemoryIn,
           cMemory := "SS2_A4_32DO_DO_Vars".DO13.cMemory,
           iCounterIn := "SS2_A4_32DO_DO_Vars".DO13.iCounterIn,
           iCounterOut := "SS2_A4_32DO_DO_Vars".DO13.iCounterOut,
           xOutput => "SS2_A4_32DO_DO_Vars".DO13.xOutput);
   "DO12.04.13" := "SS2_A4_32DO_DO_Vars".DO13.xOutput;
END_REGION

REGION Network 14: DQb5
   RUNG wire#powerrail
      "DOvar"(iFuncSystem := "SS2_A4_32DO_DO_Vars".DO14.iFuncSystemID, iFuncVar := "SS2_A4_32DO_DO_Vars".DO14.iFuncVar, xOutput => "SS2_A4_32DO_DO_Vars".DO14.xInput)
   END_RUNG
   RUNG wire#powerrail
      "DOadv"(xInput := "SS2_A4_32DO_DO_Vars".DO14.xInput, xInversion := "SS2_A4_32DO_DO_Vars".DO14.xInversion, cMOA := "SS2_A4_32DO_DO_Vars".DO14.cMOA, xMemoryOut := "SS2_A4_32DO_DO_Vars".DO14.xMemoryOut, xMemoryIn := "SS2_A4_32DO_DO_Vars".DO14.xMemoryIn, cMemory := "SS2_A4_32DO_DO_Vars".DO14.cMemory, iCounterIn := "SS2_A4_32DO_DO_Vars".DO14.iCounterIn, iCounterOut := "SS2_A4_32DO_DO_Vars".DO14.iCounterOut, xOutput => "SS2_A4_32DO_DO_Vars".DO14.xOutput)
   END_RUNG
   RUNG wire#powerrail
      Contact( "SS2_A4_32DO_DO_Vars".DO14.xOutput )
      Coil( "DO12.04.14" )
   END_RUNG
   // the same network as SCL:
   "DOvar"(iFuncSystem := "SS2_A4_32DO_DO_Vars".DO14.iFuncSystemID,
           iFuncVar := "SS2_A4_32DO_DO_Vars".DO14.iFuncVar,
           xOutput => "SS2_A4_32DO_DO_Vars".DO14.xInput);
   "DOadv"(xInput := "SS2_A4_32DO_DO_Vars".DO14.xInput,
           xInversion := "SS2_A4_32DO_DO_Vars".DO14.xInversion,
           cMOA := "SS2_A4_32DO_DO_Vars".DO14.cMOA,
           xMemoryOut := "SS2_A4_32DO_DO_Vars".DO14.xMemoryOut,
           xMemoryIn := "SS2_A4_32DO_DO_Vars".DO14.xMemoryIn,
           cMemory := "SS2_A4_32DO_DO_Vars".DO14.cMemory,
           iCounterIn := "SS2_A4_32DO_DO_Vars".DO14.iCounterIn,
           iCounterOut := "SS2_A4_32DO_DO_Vars".DO14.iCounterOut,
           xOutput => "SS2_A4_32DO_DO_Vars".DO14.xOutput);
   "DO12.04.14" := "SS2_A4_32DO_DO_Vars".DO14.xOutput;
END_REGION

REGION Network 15: DQb6
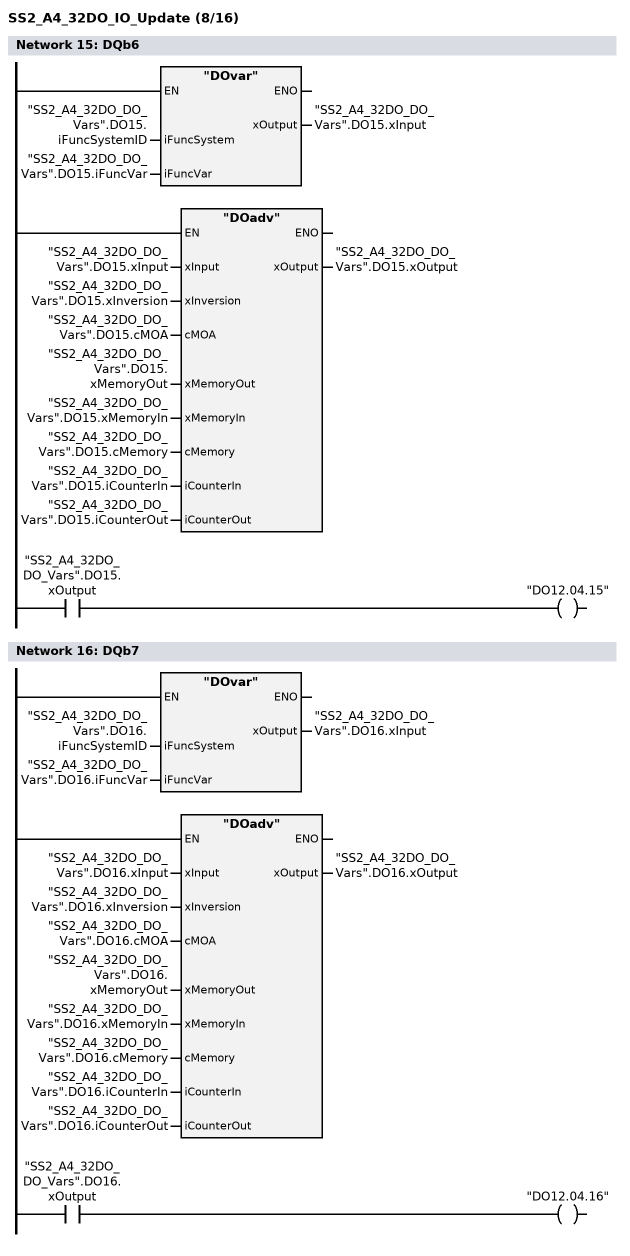
   RUNG wire#powerrail
      "DOvar"(iFuncSystem := "SS2_A4_32DO_DO_Vars".DO15.iFuncSystemID, iFuncVar := "SS2_A4_32DO_DO_Vars".DO15.iFuncVar, xOutput => "SS2_A4_32DO_DO_Vars".DO15.xInput)
   END_RUNG
   RUNG wire#powerrail
      "DOadv"(xInput := "SS2_A4_32DO_DO_Vars".DO15.xInput, xInversion := "SS2_A4_32DO_DO_Vars".DO15.xInversion, cMOA := "SS2_A4_32DO_DO_Vars".DO15.cMOA, xMemoryOut := "SS2_A4_32DO_DO_Vars".DO15.xMemoryOut, xMemoryIn := "SS2_A4_32DO_DO_Vars".DO15.xMemoryIn, cMemory := "SS2_A4_32DO_DO_Vars".DO15.cMemory, iCounterIn := "SS2_A4_32DO_DO_Vars".DO15.iCounterIn, iCounterOut := "SS2_A4_32DO_DO_Vars".DO15.iCounterOut, xOutput => "SS2_A4_32DO_DO_Vars".DO15.xOutput)
   END_RUNG
   RUNG wire#powerrail
      Contact( "SS2_A4_32DO_DO_Vars".DO15.xOutput )
      Coil( "DO12.04.15" )
   END_RUNG
   // the same network as SCL:
   "DOvar"(iFuncSystem := "SS2_A4_32DO_DO_Vars".DO15.iFuncSystemID,
           iFuncVar := "SS2_A4_32DO_DO_Vars".DO15.iFuncVar,
           xOutput => "SS2_A4_32DO_DO_Vars".DO15.xInput);
   "DOadv"(xInput := "SS2_A4_32DO_DO_Vars".DO15.xInput,
           xInversion := "SS2_A4_32DO_DO_Vars".DO15.xInversion,
           cMOA := "SS2_A4_32DO_DO_Vars".DO15.cMOA,
           xMemoryOut := "SS2_A4_32DO_DO_Vars".DO15.xMemoryOut,
           xMemoryIn := "SS2_A4_32DO_DO_Vars".DO15.xMemoryIn,
           cMemory := "SS2_A4_32DO_DO_Vars".DO15.cMemory,
           iCounterIn := "SS2_A4_32DO_DO_Vars".DO15.iCounterIn,
           iCounterOut := "SS2_A4_32DO_DO_Vars".DO15.iCounterOut,
           xOutput => "SS2_A4_32DO_DO_Vars".DO15.xOutput);
   "DO12.04.15" := "SS2_A4_32DO_DO_Vars".DO15.xOutput;
END_REGION

REGION Network 16: DQb7
   RUNG wire#powerrail
      "DOvar"(iFuncSystem := "SS2_A4_32DO_DO_Vars".DO16.iFuncSystemID, iFuncVar := "SS2_A4_32DO_DO_Vars".DO16.iFuncVar, xOutput => "SS2_A4_32DO_DO_Vars".DO16.xInput)
   END_RUNG
   RUNG wire#powerrail
      "DOadv"(xInput := "SS2_A4_32DO_DO_Vars".DO16.xInput, xInversion := "SS2_A4_32DO_DO_Vars".DO16.xInversion, cMOA := "SS2_A4_32DO_DO_Vars".DO16.cMOA, xMemoryOut := "SS2_A4_32DO_DO_Vars".DO16.xMemoryOut, xMemoryIn := "SS2_A4_32DO_DO_Vars".DO16.xMemoryIn, cMemory := "SS2_A4_32DO_DO_Vars".DO16.cMemory, iCounterIn := "SS2_A4_32DO_DO_Vars".DO16.iCounterIn, iCounterOut := "SS2_A4_32DO_DO_Vars".DO16.iCounterOut, xOutput => "SS2_A4_32DO_DO_Vars".DO16.xOutput)
   END_RUNG
   RUNG wire#powerrail
      Contact( "SS2_A4_32DO_DO_Vars".DO16.xOutput )
      Coil( "DO12.04.16" )
   END_RUNG
   // the same network as SCL:
   "DOvar"(iFuncSystem := "SS2_A4_32DO_DO_Vars".DO16.iFuncSystemID,
           iFuncVar := "SS2_A4_32DO_DO_Vars".DO16.iFuncVar,
           xOutput => "SS2_A4_32DO_DO_Vars".DO16.xInput);
   "DOadv"(xInput := "SS2_A4_32DO_DO_Vars".DO16.xInput,
           xInversion := "SS2_A4_32DO_DO_Vars".DO16.xInversion,
           cMOA := "SS2_A4_32DO_DO_Vars".DO16.cMOA,
           xMemoryOut := "SS2_A4_32DO_DO_Vars".DO16.xMemoryOut,
           xMemoryIn := "SS2_A4_32DO_DO_Vars".DO16.xMemoryIn,
           cMemory := "SS2_A4_32DO_DO_Vars".DO16.cMemory,
           iCounterIn := "SS2_A4_32DO_DO_Vars".DO16.iCounterIn,
           iCounterOut := "SS2_A4_32DO_DO_Vars".DO16.iCounterOut,
           xOutput => "SS2_A4_32DO_DO_Vars".DO16.xOutput);
   "DO12.04.16" := "SS2_A4_32DO_DO_Vars".DO16.xOutput;
END_REGION

REGION Network 17: DQc0
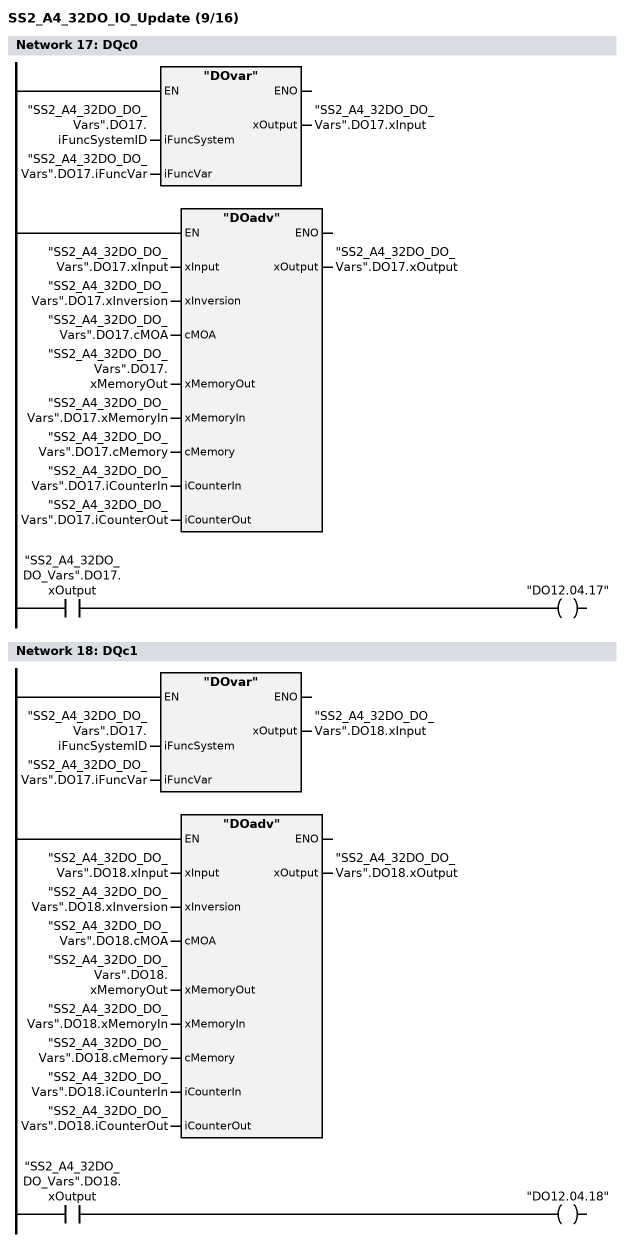
   RUNG wire#powerrail
      "DOvar"(iFuncSystem := "SS2_A4_32DO_DO_Vars".DO17.iFuncSystemID, iFuncVar := "SS2_A4_32DO_DO_Vars".DO17.iFuncVar, xOutput => "SS2_A4_32DO_DO_Vars".DO17.xInput)
   END_RUNG
   RUNG wire#powerrail
      "DOadv"(xInput := "SS2_A4_32DO_DO_Vars".DO17.xInput, xInversion := "SS2_A4_32DO_DO_Vars".DO17.xInversion, cMOA := "SS2_A4_32DO_DO_Vars".DO17.cMOA, xMemoryOut := "SS2_A4_32DO_DO_Vars".DO17.xMemoryOut, xMemoryIn := "SS2_A4_32DO_DO_Vars".DO17.xMemoryIn, cMemory := "SS2_A4_32DO_DO_Vars".DO17.cMemory, iCounterIn := "SS2_A4_32DO_DO_Vars".DO17.iCounterIn, iCounterOut := "SS2_A4_32DO_DO_Vars".DO17.iCounterOut, xOutput => "SS2_A4_32DO_DO_Vars".DO17.xOutput)
   END_RUNG
   RUNG wire#powerrail
      Contact( "SS2_A4_32DO_DO_Vars".DO17.xOutput )
      Coil( "DO12.04.17" )
   END_RUNG
   // the same network as SCL:
   "DOvar"(iFuncSystem := "SS2_A4_32DO_DO_Vars".DO17.iFuncSystemID,
           iFuncVar := "SS2_A4_32DO_DO_Vars".DO17.iFuncVar,
           xOutput => "SS2_A4_32DO_DO_Vars".DO17.xInput);
   "DOadv"(xInput := "SS2_A4_32DO_DO_Vars".DO17.xInput,
           xInversion := "SS2_A4_32DO_DO_Vars".DO17.xInversion,
           cMOA := "SS2_A4_32DO_DO_Vars".DO17.cMOA,
           xMemoryOut := "SS2_A4_32DO_DO_Vars".DO17.xMemoryOut,
           xMemoryIn := "SS2_A4_32DO_DO_Vars".DO17.xMemoryIn,
           cMemory := "SS2_A4_32DO_DO_Vars".DO17.cMemory,
           iCounterIn := "SS2_A4_32DO_DO_Vars".DO17.iCounterIn,
           iCounterOut := "SS2_A4_32DO_DO_Vars".DO17.iCounterOut,
           xOutput => "SS2_A4_32DO_DO_Vars".DO17.xOutput);
   "DO12.04.17" := "SS2_A4_32DO_DO_Vars".DO17.xOutput;
END_REGION

REGION Network 18: DQc1
   RUNG wire#powerrail
      "DOvar"(iFuncSystem := "SS2_A4_32DO_DO_Vars".DO17.iFuncSystemID, iFuncVar := "SS2_A4_32DO_DO_Vars".DO17.iFuncVar, xOutput => "SS2_A4_32DO_DO_Vars".DO18.xInput)
   END_RUNG
   RUNG wire#powerrail
      "DOadv"(xInput := "SS2_A4_32DO_DO_Vars".DO18.xInput, xInversion := "SS2_A4_32DO_DO_Vars".DO18.xInversion, cMOA := "SS2_A4_32DO_DO_Vars".DO18.cMOA, xMemoryOut := "SS2_A4_32DO_DO_Vars".DO18.xMemoryOut, xMemoryIn := "SS2_A4_32DO_DO_Vars".DO18.xMemoryIn, cMemory := "SS2_A4_32DO_DO_Vars".DO18.cMemory, iCounterIn := "SS2_A4_32DO_DO_Vars".DO18.iCounterIn, iCounterOut := "SS2_A4_32DO_DO_Vars".DO18.iCounterOut, xOutput => "SS2_A4_32DO_DO_Vars".DO18.xOutput)
   END_RUNG
   RUNG wire#powerrail
      Contact( "SS2_A4_32DO_DO_Vars".DO18.xOutput )
      Coil( "DO12.04.18" )
   END_RUNG
   // the same network as SCL:
   "DOvar"(iFuncSystem := "SS2_A4_32DO_DO_Vars".DO17.iFuncSystemID,
           iFuncVar := "SS2_A4_32DO_DO_Vars".DO17.iFuncVar,
           xOutput => "SS2_A4_32DO_DO_Vars".DO18.xInput);
   "DOadv"(xInput := "SS2_A4_32DO_DO_Vars".DO18.xInput,
           xInversion := "SS2_A4_32DO_DO_Vars".DO18.xInversion,
           cMOA := "SS2_A4_32DO_DO_Vars".DO18.cMOA,
           xMemoryOut := "SS2_A4_32DO_DO_Vars".DO18.xMemoryOut,
           xMemoryIn := "SS2_A4_32DO_DO_Vars".DO18.xMemoryIn,
           cMemory := "SS2_A4_32DO_DO_Vars".DO18.cMemory,
           iCounterIn := "SS2_A4_32DO_DO_Vars".DO18.iCounterIn,
           iCounterOut := "SS2_A4_32DO_DO_Vars".DO18.iCounterOut,
           xOutput => "SS2_A4_32DO_DO_Vars".DO18.xOutput);
   "DO12.04.18" := "SS2_A4_32DO_DO_Vars".DO18.xOutput;
END_REGION

REGION Network 19: DQc2
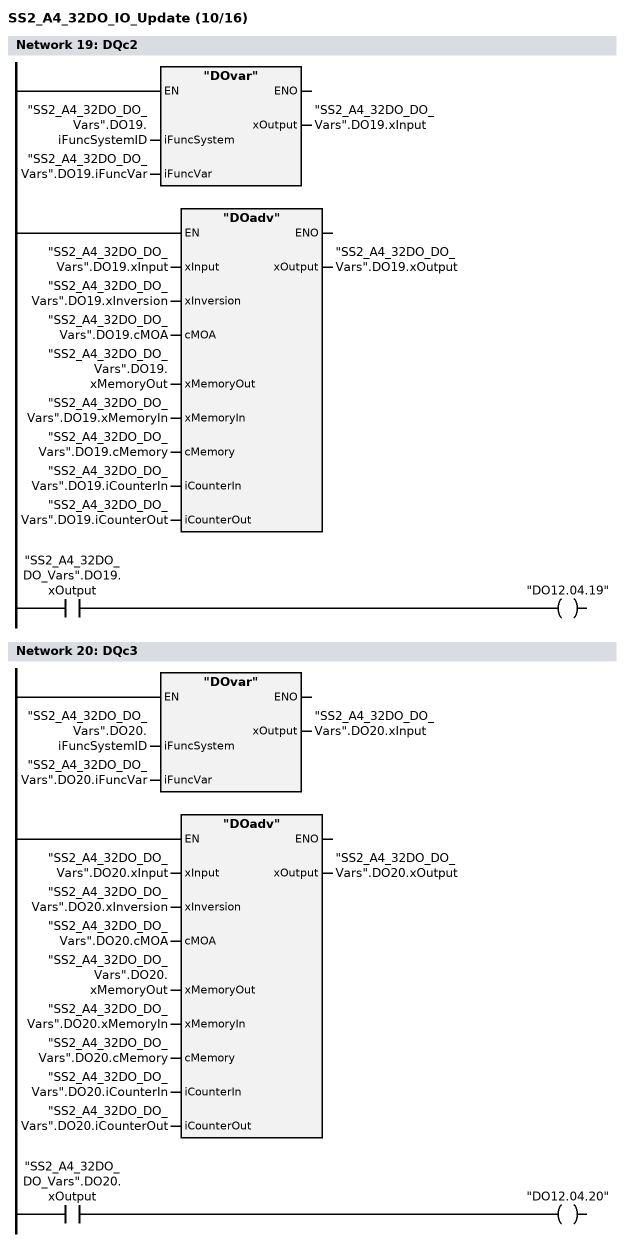
   RUNG wire#powerrail
      "DOvar"(iFuncSystem := "SS2_A4_32DO_DO_Vars".DO19.iFuncSystemID, iFuncVar := "SS2_A4_32DO_DO_Vars".DO19.iFuncVar, xOutput => "SS2_A4_32DO_DO_Vars".DO19.xInput)
   END_RUNG
   RUNG wire#powerrail
      "DOadv"(xInput := "SS2_A4_32DO_DO_Vars".DO19.xInput, xInversion := "SS2_A4_32DO_DO_Vars".DO19.xInversion, cMOA := "SS2_A4_32DO_DO_Vars".DO19.cMOA, xMemoryOut := "SS2_A4_32DO_DO_Vars".DO19.xMemoryOut, xMemoryIn := "SS2_A4_32DO_DO_Vars".DO19.xMemoryIn, cMemory := "SS2_A4_32DO_DO_Vars".DO19.cMemory, iCounterIn := "SS2_A4_32DO_DO_Vars".DO19.iCounterIn, iCounterOut := "SS2_A4_32DO_DO_Vars".DO19.iCounterOut, xOutput => "SS2_A4_32DO_DO_Vars".DO19.xOutput)
   END_RUNG
   RUNG wire#powerrail
      Contact( "SS2_A4_32DO_DO_Vars".DO19.xOutput )
      Coil( "DO12.04.19" )
   END_RUNG
   // the same network as SCL:
   "DOvar"(iFuncSystem := "SS2_A4_32DO_DO_Vars".DO19.iFuncSystemID,
           iFuncVar := "SS2_A4_32DO_DO_Vars".DO19.iFuncVar,
           xOutput => "SS2_A4_32DO_DO_Vars".DO19.xInput);
   "DOadv"(xInput := "SS2_A4_32DO_DO_Vars".DO19.xInput,
           xInversion := "SS2_A4_32DO_DO_Vars".DO19.xInversion,
           cMOA := "SS2_A4_32DO_DO_Vars".DO19.cMOA,
           xMemoryOut := "SS2_A4_32DO_DO_Vars".DO19.xMemoryOut,
           xMemoryIn := "SS2_A4_32DO_DO_Vars".DO19.xMemoryIn,
           cMemory := "SS2_A4_32DO_DO_Vars".DO19.cMemory,
           iCounterIn := "SS2_A4_32DO_DO_Vars".DO19.iCounterIn,
           iCounterOut := "SS2_A4_32DO_DO_Vars".DO19.iCounterOut,
           xOutput => "SS2_A4_32DO_DO_Vars".DO19.xOutput);
   "DO12.04.19" := "SS2_A4_32DO_DO_Vars".DO19.xOutput;
END_REGION

REGION Network 20: DQc3
   RUNG wire#powerrail
      "DOvar"(iFuncSystem := "SS2_A4_32DO_DO_Vars".DO20.iFuncSystemID, iFuncVar := "SS2_A4_32DO_DO_Vars".DO20.iFuncVar, xOutput => "SS2_A4_32DO_DO_Vars".DO20.xInput)
   END_RUNG
   RUNG wire#powerrail
      "DOadv"(xInput := "SS2_A4_32DO_DO_Vars".DO20.xInput, xInversion := "SS2_A4_32DO_DO_Vars".DO20.xInversion, cMOA := "SS2_A4_32DO_DO_Vars".DO20.cMOA, xMemoryOut := "SS2_A4_32DO_DO_Vars".DO20.xMemoryOut, xMemoryIn := "SS2_A4_32DO_DO_Vars".DO20.xMemoryIn, cMemory := "SS2_A4_32DO_DO_Vars".DO20.cMemory, iCounterIn := "SS2_A4_32DO_DO_Vars".DO20.iCounterIn, iCounterOut := "SS2_A4_32DO_DO_Vars".DO20.iCounterOut, xOutput => "SS2_A4_32DO_DO_Vars".DO20.xOutput)
   END_RUNG
   RUNG wire#powerrail
      Contact( "SS2_A4_32DO_DO_Vars".DO20.xOutput )
      Coil( "DO12.04.20" )
   END_RUNG
   // the same network as SCL:
   "DOvar"(iFuncSystem := "SS2_A4_32DO_DO_Vars".DO20.iFuncSystemID,
           iFuncVar := "SS2_A4_32DO_DO_Vars".DO20.iFuncVar,
           xOutput => "SS2_A4_32DO_DO_Vars".DO20.xInput);
   "DOadv"(xInput := "SS2_A4_32DO_DO_Vars".DO20.xInput,
           xInversion := "SS2_A4_32DO_DO_Vars".DO20.xInversion,
           cMOA := "SS2_A4_32DO_DO_Vars".DO20.cMOA,
           xMemoryOut := "SS2_A4_32DO_DO_Vars".DO20.xMemoryOut,
           xMemoryIn := "SS2_A4_32DO_DO_Vars".DO20.xMemoryIn,
           cMemory := "SS2_A4_32DO_DO_Vars".DO20.cMemory,
           iCounterIn := "SS2_A4_32DO_DO_Vars".DO20.iCounterIn,
           iCounterOut := "SS2_A4_32DO_DO_Vars".DO20.iCounterOut,
           xOutput => "SS2_A4_32DO_DO_Vars".DO20.xOutput);
   "DO12.04.20" := "SS2_A4_32DO_DO_Vars".DO20.xOutput;
END_REGION

REGION Network 21: DQc4
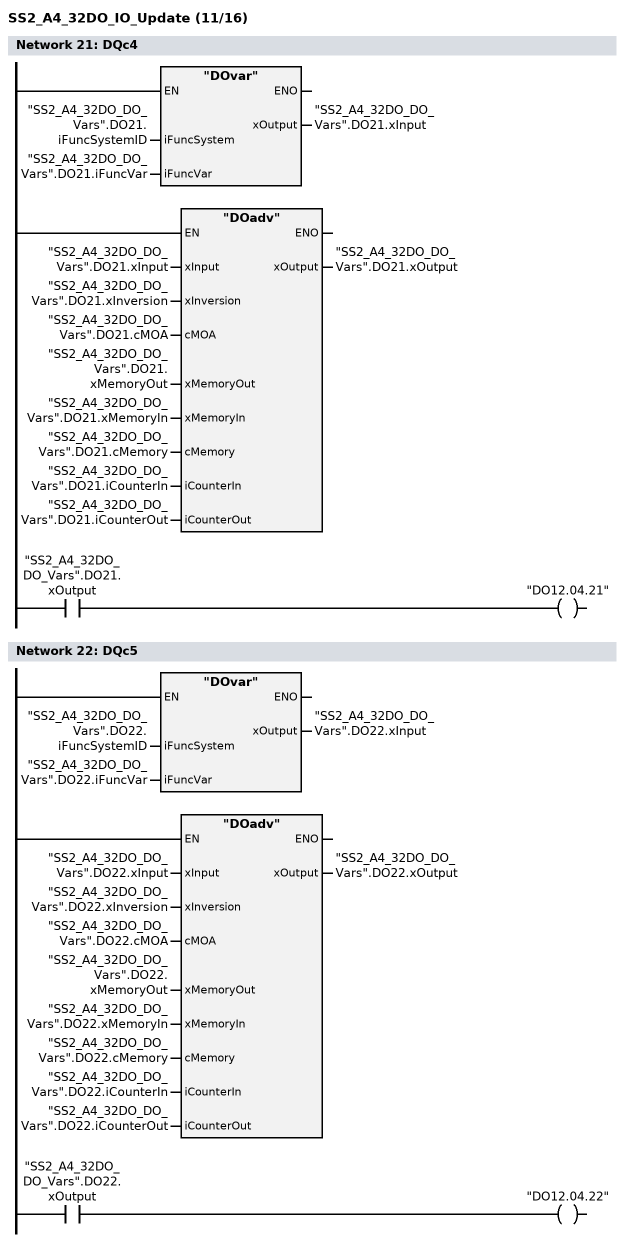
   RUNG wire#powerrail
      "DOvar"(iFuncSystem := "SS2_A4_32DO_DO_Vars".DO21.iFuncSystemID, iFuncVar := "SS2_A4_32DO_DO_Vars".DO21.iFuncVar, xOutput => "SS2_A4_32DO_DO_Vars".DO21.xInput)
   END_RUNG
   RUNG wire#powerrail
      "DOadv"(xInput := "SS2_A4_32DO_DO_Vars".DO21.xInput, xInversion := "SS2_A4_32DO_DO_Vars".DO21.xInversion, cMOA := "SS2_A4_32DO_DO_Vars".DO21.cMOA, xMemoryOut := "SS2_A4_32DO_DO_Vars".DO21.xMemoryOut, xMemoryIn := "SS2_A4_32DO_DO_Vars".DO21.xMemoryIn, cMemory := "SS2_A4_32DO_DO_Vars".DO21.cMemory, iCounterIn := "SS2_A4_32DO_DO_Vars".DO21.iCounterIn, iCounterOut := "SS2_A4_32DO_DO_Vars".DO21.iCounterOut, xOutput => "SS2_A4_32DO_DO_Vars".DO21.xOutput)
   END_RUNG
   RUNG wire#powerrail
      Contact( "SS2_A4_32DO_DO_Vars".DO21.xOutput )
      Coil( "DO12.04.21" )
   END_RUNG
   // the same network as SCL:
   "DOvar"(iFuncSystem := "SS2_A4_32DO_DO_Vars".DO21.iFuncSystemID,
           iFuncVar := "SS2_A4_32DO_DO_Vars".DO21.iFuncVar,
           xOutput => "SS2_A4_32DO_DO_Vars".DO21.xInput);
   "DOadv"(xInput := "SS2_A4_32DO_DO_Vars".DO21.xInput,
           xInversion := "SS2_A4_32DO_DO_Vars".DO21.xInversion,
           cMOA := "SS2_A4_32DO_DO_Vars".DO21.cMOA,
           xMemoryOut := "SS2_A4_32DO_DO_Vars".DO21.xMemoryOut,
           xMemoryIn := "SS2_A4_32DO_DO_Vars".DO21.xMemoryIn,
           cMemory := "SS2_A4_32DO_DO_Vars".DO21.cMemory,
           iCounterIn := "SS2_A4_32DO_DO_Vars".DO21.iCounterIn,
           iCounterOut := "SS2_A4_32DO_DO_Vars".DO21.iCounterOut,
           xOutput => "SS2_A4_32DO_DO_Vars".DO21.xOutput);
   "DO12.04.21" := "SS2_A4_32DO_DO_Vars".DO21.xOutput;
END_REGION

REGION Network 22: DQc5
   RUNG wire#powerrail
      "DOvar"(iFuncSystem := "SS2_A4_32DO_DO_Vars".DO22.iFuncSystemID, iFuncVar := "SS2_A4_32DO_DO_Vars".DO22.iFuncVar, xOutput => "SS2_A4_32DO_DO_Vars".DO22.xInput)
   END_RUNG
   RUNG wire#powerrail
      "DOadv"(xInput := "SS2_A4_32DO_DO_Vars".DO22.xInput, xInversion := "SS2_A4_32DO_DO_Vars".DO22.xInversion, cMOA := "SS2_A4_32DO_DO_Vars".DO22.cMOA, xMemoryOut := "SS2_A4_32DO_DO_Vars".DO22.xMemoryOut, xMemoryIn := "SS2_A4_32DO_DO_Vars".DO22.xMemoryIn, cMemory := "SS2_A4_32DO_DO_Vars".DO22.cMemory, iCounterIn := "SS2_A4_32DO_DO_Vars".DO22.iCounterIn, iCounterOut := "SS2_A4_32DO_DO_Vars".DO22.iCounterOut, xOutput => "SS2_A4_32DO_DO_Vars".DO22.xOutput)
   END_RUNG
   RUNG wire#powerrail
      Contact( "SS2_A4_32DO_DO_Vars".DO22.xOutput )
      Coil( "DO12.04.22" )
   END_RUNG
   // the same network as SCL:
   "DOvar"(iFuncSystem := "SS2_A4_32DO_DO_Vars".DO22.iFuncSystemID,
           iFuncVar := "SS2_A4_32DO_DO_Vars".DO22.iFuncVar,
           xOutput => "SS2_A4_32DO_DO_Vars".DO22.xInput);
   "DOadv"(xInput := "SS2_A4_32DO_DO_Vars".DO22.xInput,
           xInversion := "SS2_A4_32DO_DO_Vars".DO22.xInversion,
           cMOA := "SS2_A4_32DO_DO_Vars".DO22.cMOA,
           xMemoryOut := "SS2_A4_32DO_DO_Vars".DO22.xMemoryOut,
           xMemoryIn := "SS2_A4_32DO_DO_Vars".DO22.xMemoryIn,
           cMemory := "SS2_A4_32DO_DO_Vars".DO22.cMemory,
           iCounterIn := "SS2_A4_32DO_DO_Vars".DO22.iCounterIn,
           iCounterOut := "SS2_A4_32DO_DO_Vars".DO22.iCounterOut,
           xOutput => "SS2_A4_32DO_DO_Vars".DO22.xOutput);
   "DO12.04.22" := "SS2_A4_32DO_DO_Vars".DO22.xOutput;
END_REGION

REGION Network 23: DQc6
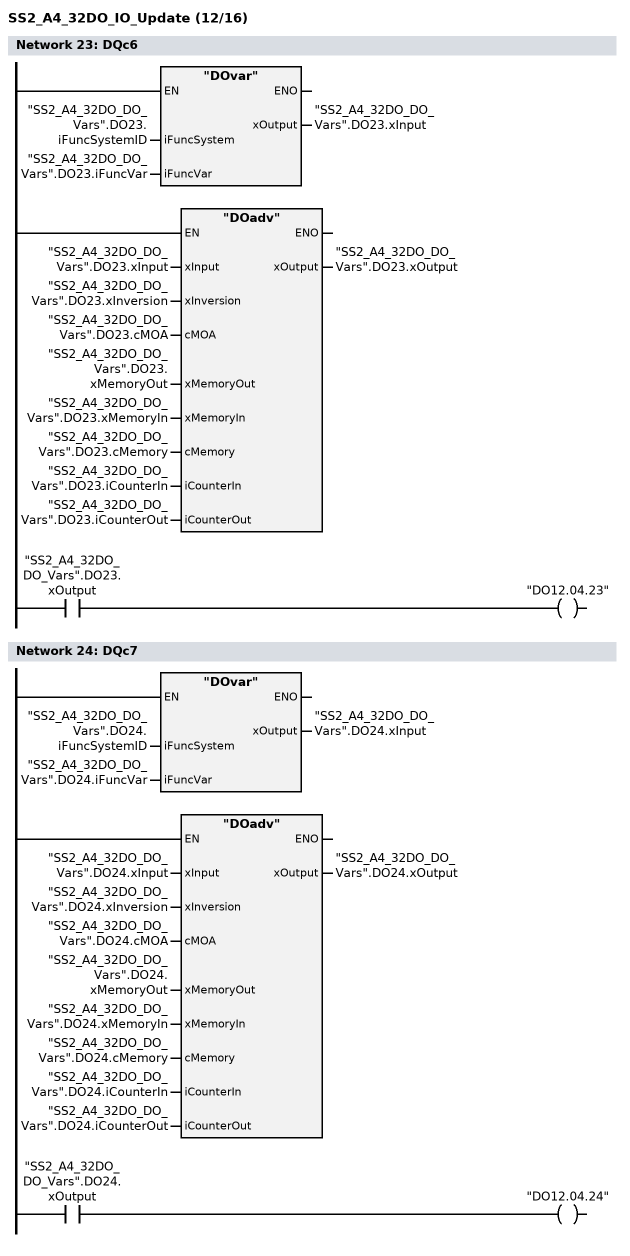
   RUNG wire#powerrail
      "DOvar"(iFuncSystem := "SS2_A4_32DO_DO_Vars".DO23.iFuncSystemID, iFuncVar := "SS2_A4_32DO_DO_Vars".DO23.iFuncVar, xOutput => "SS2_A4_32DO_DO_Vars".DO23.xInput)
   END_RUNG
   RUNG wire#powerrail
      "DOadv"(xInput := "SS2_A4_32DO_DO_Vars".DO23.xInput, xInversion := "SS2_A4_32DO_DO_Vars".DO23.xInversion, cMOA := "SS2_A4_32DO_DO_Vars".DO23.cMOA, xMemoryOut := "SS2_A4_32DO_DO_Vars".DO23.xMemoryOut, xMemoryIn := "SS2_A4_32DO_DO_Vars".DO23.xMemoryIn, cMemory := "SS2_A4_32DO_DO_Vars".DO23.cMemory, iCounterIn := "SS2_A4_32DO_DO_Vars".DO23.iCounterIn, iCounterOut := "SS2_A4_32DO_DO_Vars".DO23.iCounterOut, xOutput => "SS2_A4_32DO_DO_Vars".DO23.xOutput)
   END_RUNG
   RUNG wire#powerrail
      Contact( "SS2_A4_32DO_DO_Vars".DO23.xOutput )
      Coil( "DO12.04.23" )
   END_RUNG
   // the same network as SCL:
   "DOvar"(iFuncSystem := "SS2_A4_32DO_DO_Vars".DO23.iFuncSystemID,
           iFuncVar := "SS2_A4_32DO_DO_Vars".DO23.iFuncVar,
           xOutput => "SS2_A4_32DO_DO_Vars".DO23.xInput);
   "DOadv"(xInput := "SS2_A4_32DO_DO_Vars".DO23.xInput,
           xInversion := "SS2_A4_32DO_DO_Vars".DO23.xInversion,
           cMOA := "SS2_A4_32DO_DO_Vars".DO23.cMOA,
           xMemoryOut := "SS2_A4_32DO_DO_Vars".DO23.xMemoryOut,
           xMemoryIn := "SS2_A4_32DO_DO_Vars".DO23.xMemoryIn,
           cMemory := "SS2_A4_32DO_DO_Vars".DO23.cMemory,
           iCounterIn := "SS2_A4_32DO_DO_Vars".DO23.iCounterIn,
           iCounterOut := "SS2_A4_32DO_DO_Vars".DO23.iCounterOut,
           xOutput => "SS2_A4_32DO_DO_Vars".DO23.xOutput);
   "DO12.04.23" := "SS2_A4_32DO_DO_Vars".DO23.xOutput;
END_REGION

REGION Network 24: DQc7
   RUNG wire#powerrail
      "DOvar"(iFuncSystem := "SS2_A4_32DO_DO_Vars".DO24.iFuncSystemID, iFuncVar := "SS2_A4_32DO_DO_Vars".DO24.iFuncVar, xOutput => "SS2_A4_32DO_DO_Vars".DO24.xInput)
   END_RUNG
   RUNG wire#powerrail
      "DOadv"(xInput := "SS2_A4_32DO_DO_Vars".DO24.xInput, xInversion := "SS2_A4_32DO_DO_Vars".DO24.xInversion, cMOA := "SS2_A4_32DO_DO_Vars".DO24.cMOA, xMemoryOut := "SS2_A4_32DO_DO_Vars".DO24.xMemoryOut, xMemoryIn := "SS2_A4_32DO_DO_Vars".DO24.xMemoryIn, cMemory := "SS2_A4_32DO_DO_Vars".DO24.cMemory, iCounterIn := "SS2_A4_32DO_DO_Vars".DO24.iCounterIn, iCounterOut := "SS2_A4_32DO_DO_Vars".DO24.iCounterOut, xOutput => "SS2_A4_32DO_DO_Vars".DO24.xOutput)
   END_RUNG
   RUNG wire#powerrail
      Contact( "SS2_A4_32DO_DO_Vars".DO24.xOutput )
      Coil( "DO12.04.24" )
   END_RUNG
   // the same network as SCL:
   "DOvar"(iFuncSystem := "SS2_A4_32DO_DO_Vars".DO24.iFuncSystemID,
           iFuncVar := "SS2_A4_32DO_DO_Vars".DO24.iFuncVar,
           xOutput => "SS2_A4_32DO_DO_Vars".DO24.xInput);
   "DOadv"(xInput := "SS2_A4_32DO_DO_Vars".DO24.xInput,
           xInversion := "SS2_A4_32DO_DO_Vars".DO24.xInversion,
           cMOA := "SS2_A4_32DO_DO_Vars".DO24.cMOA,
           xMemoryOut := "SS2_A4_32DO_DO_Vars".DO24.xMemoryOut,
           xMemoryIn := "SS2_A4_32DO_DO_Vars".DO24.xMemoryIn,
           cMemory := "SS2_A4_32DO_DO_Vars".DO24.cMemory,
           iCounterIn := "SS2_A4_32DO_DO_Vars".DO24.iCounterIn,
           iCounterOut := "SS2_A4_32DO_DO_Vars".DO24.iCounterOut,
           xOutput => "SS2_A4_32DO_DO_Vars".DO24.xOutput);
   "DO12.04.24" := "SS2_A4_32DO_DO_Vars".DO24.xOutput;
END_REGION

REGION Network 25: DQd0
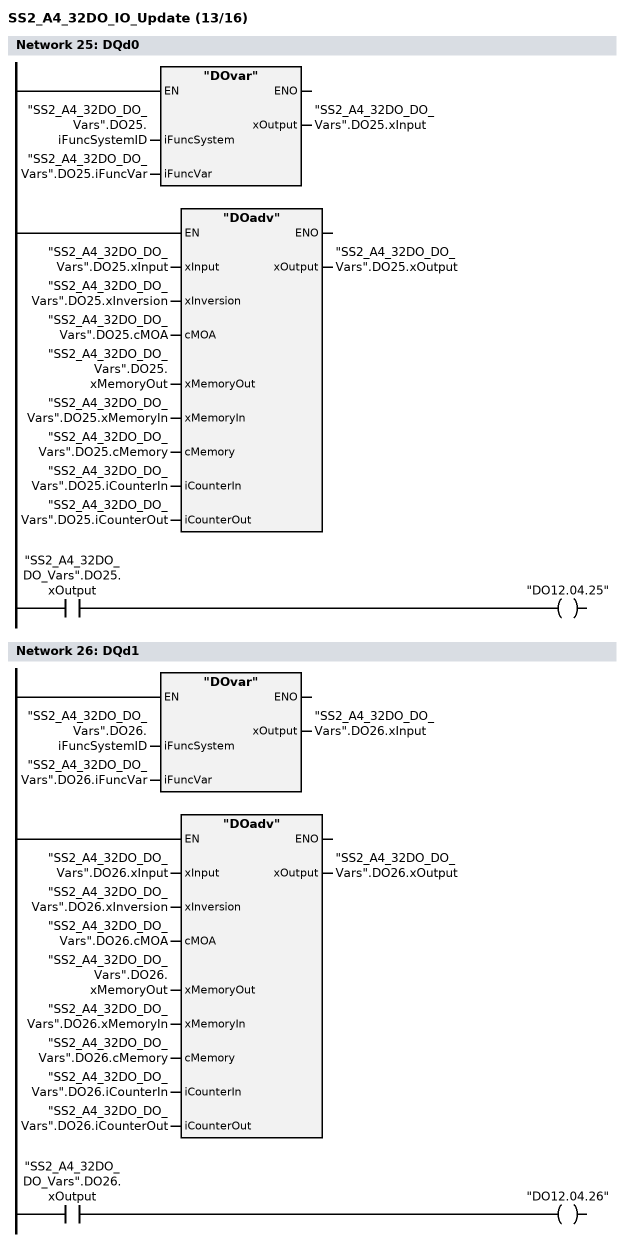
   RUNG wire#powerrail
      "DOvar"(iFuncSystem := "SS2_A4_32DO_DO_Vars".DO25.iFuncSystemID, iFuncVar := "SS2_A4_32DO_DO_Vars".DO25.iFuncVar, xOutput => "SS2_A4_32DO_DO_Vars".DO25.xInput)
   END_RUNG
   RUNG wire#powerrail
      "DOadv"(xInput := "SS2_A4_32DO_DO_Vars".DO25.xInput, xInversion := "SS2_A4_32DO_DO_Vars".DO25.xInversion, cMOA := "SS2_A4_32DO_DO_Vars".DO25.cMOA, xMemoryOut := "SS2_A4_32DO_DO_Vars".DO25.xMemoryOut, xMemoryIn := "SS2_A4_32DO_DO_Vars".DO25.xMemoryIn, cMemory := "SS2_A4_32DO_DO_Vars".DO25.cMemory, iCounterIn := "SS2_A4_32DO_DO_Vars".DO25.iCounterIn, iCounterOut := "SS2_A4_32DO_DO_Vars".DO25.iCounterOut, xOutput => "SS2_A4_32DO_DO_Vars".DO25.xOutput)
   END_RUNG
   RUNG wire#powerrail
      Contact( "SS2_A4_32DO_DO_Vars".DO25.xOutput )
      Coil( "DO12.04.25" )
   END_RUNG
   // the same network as SCL:
   "DOvar"(iFuncSystem := "SS2_A4_32DO_DO_Vars".DO25.iFuncSystemID,
           iFuncVar := "SS2_A4_32DO_DO_Vars".DO25.iFuncVar,
           xOutput => "SS2_A4_32DO_DO_Vars".DO25.xInput);
   "DOadv"(xInput := "SS2_A4_32DO_DO_Vars".DO25.xInput,
           xInversion := "SS2_A4_32DO_DO_Vars".DO25.xInversion,
           cMOA := "SS2_A4_32DO_DO_Vars".DO25.cMOA,
           xMemoryOut := "SS2_A4_32DO_DO_Vars".DO25.xMemoryOut,
           xMemoryIn := "SS2_A4_32DO_DO_Vars".DO25.xMemoryIn,
           cMemory := "SS2_A4_32DO_DO_Vars".DO25.cMemory,
           iCounterIn := "SS2_A4_32DO_DO_Vars".DO25.iCounterIn,
           iCounterOut := "SS2_A4_32DO_DO_Vars".DO25.iCounterOut,
           xOutput => "SS2_A4_32DO_DO_Vars".DO25.xOutput);
   "DO12.04.25" := "SS2_A4_32DO_DO_Vars".DO25.xOutput;
END_REGION

REGION Network 26: DQd1
   RUNG wire#powerrail
      "DOvar"(iFuncSystem := "SS2_A4_32DO_DO_Vars".DO26.iFuncSystemID, iFuncVar := "SS2_A4_32DO_DO_Vars".DO26.iFuncVar, xOutput => "SS2_A4_32DO_DO_Vars".DO26.xInput)
   END_RUNG
   RUNG wire#powerrail
      "DOadv"(xInput := "SS2_A4_32DO_DO_Vars".DO26.xInput, xInversion := "SS2_A4_32DO_DO_Vars".DO26.xInversion, cMOA := "SS2_A4_32DO_DO_Vars".DO26.cMOA, xMemoryOut := "SS2_A4_32DO_DO_Vars".DO26.xMemoryOut, xMemoryIn := "SS2_A4_32DO_DO_Vars".DO26.xMemoryIn, cMemory := "SS2_A4_32DO_DO_Vars".DO26.cMemory, iCounterIn := "SS2_A4_32DO_DO_Vars".DO26.iCounterIn, iCounterOut := "SS2_A4_32DO_DO_Vars".DO26.iCounterOut, xOutput => "SS2_A4_32DO_DO_Vars".DO26.xOutput)
   END_RUNG
   RUNG wire#powerrail
      Contact( "SS2_A4_32DO_DO_Vars".DO26.xOutput )
      Coil( "DO12.04.26" )
   END_RUNG
   // the same network as SCL:
   "DOvar"(iFuncSystem := "SS2_A4_32DO_DO_Vars".DO26.iFuncSystemID,
           iFuncVar := "SS2_A4_32DO_DO_Vars".DO26.iFuncVar,
           xOutput => "SS2_A4_32DO_DO_Vars".DO26.xInput);
   "DOadv"(xInput := "SS2_A4_32DO_DO_Vars".DO26.xInput,
           xInversion := "SS2_A4_32DO_DO_Vars".DO26.xInversion,
           cMOA := "SS2_A4_32DO_DO_Vars".DO26.cMOA,
           xMemoryOut := "SS2_A4_32DO_DO_Vars".DO26.xMemoryOut,
           xMemoryIn := "SS2_A4_32DO_DO_Vars".DO26.xMemoryIn,
           cMemory := "SS2_A4_32DO_DO_Vars".DO26.cMemory,
           iCounterIn := "SS2_A4_32DO_DO_Vars".DO26.iCounterIn,
           iCounterOut := "SS2_A4_32DO_DO_Vars".DO26.iCounterOut,
           xOutput => "SS2_A4_32DO_DO_Vars".DO26.xOutput);
   "DO12.04.26" := "SS2_A4_32DO_DO_Vars".DO26.xOutput;
END_REGION

REGION Network 27: DQd2
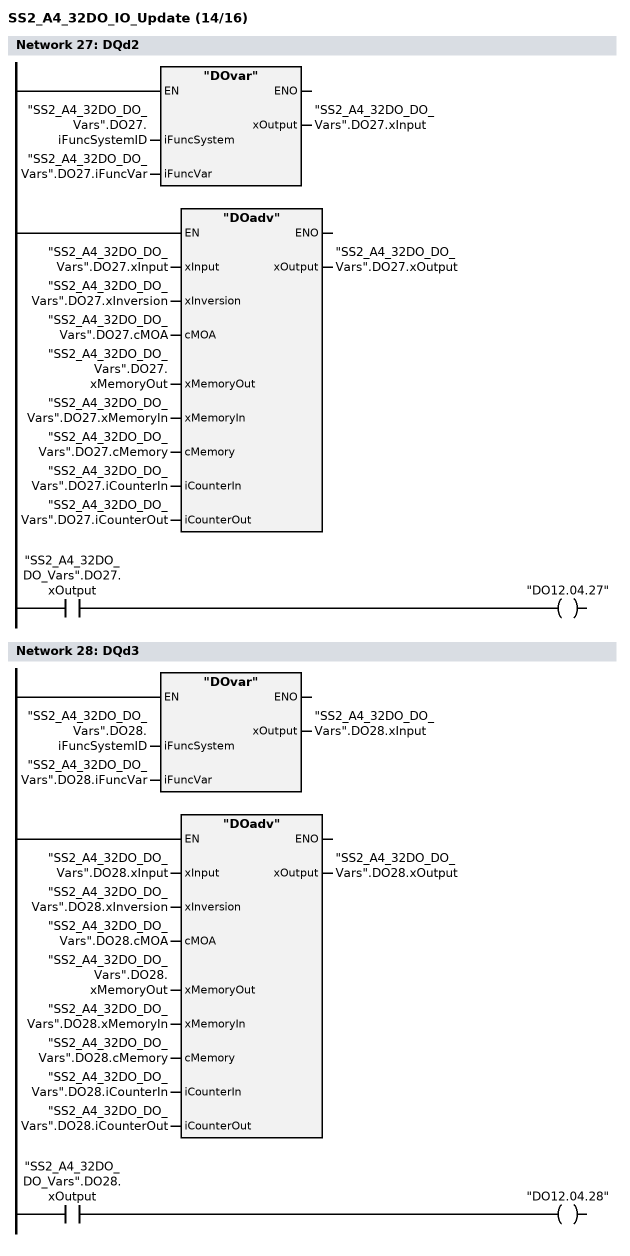
   RUNG wire#powerrail
      "DOvar"(iFuncSystem := "SS2_A4_32DO_DO_Vars".DO27.iFuncSystemID, iFuncVar := "SS2_A4_32DO_DO_Vars".DO27.iFuncVar, xOutput => "SS2_A4_32DO_DO_Vars".DO27.xInput)
   END_RUNG
   RUNG wire#powerrail
      "DOadv"(xInput := "SS2_A4_32DO_DO_Vars".DO27.xInput, xInversion := "SS2_A4_32DO_DO_Vars".DO27.xInversion, cMOA := "SS2_A4_32DO_DO_Vars".DO27.cMOA, xMemoryOut := "SS2_A4_32DO_DO_Vars".DO27.xMemoryOut, xMemoryIn := "SS2_A4_32DO_DO_Vars".DO27.xMemoryIn, cMemory := "SS2_A4_32DO_DO_Vars".DO27.cMemory, iCounterIn := "SS2_A4_32DO_DO_Vars".DO27.iCounterIn, iCounterOut := "SS2_A4_32DO_DO_Vars".DO27.iCounterOut, xOutput => "SS2_A4_32DO_DO_Vars".DO27.xOutput)
   END_RUNG
   RUNG wire#powerrail
      Contact( "SS2_A4_32DO_DO_Vars".DO27.xOutput )
      Coil( "DO12.04.27" )
   END_RUNG
   // the same network as SCL:
   "DOvar"(iFuncSystem := "SS2_A4_32DO_DO_Vars".DO27.iFuncSystemID,
           iFuncVar := "SS2_A4_32DO_DO_Vars".DO27.iFuncVar,
           xOutput => "SS2_A4_32DO_DO_Vars".DO27.xInput);
   "DOadv"(xInput := "SS2_A4_32DO_DO_Vars".DO27.xInput,
           xInversion := "SS2_A4_32DO_DO_Vars".DO27.xInversion,
           cMOA := "SS2_A4_32DO_DO_Vars".DO27.cMOA,
           xMemoryOut := "SS2_A4_32DO_DO_Vars".DO27.xMemoryOut,
           xMemoryIn := "SS2_A4_32DO_DO_Vars".DO27.xMemoryIn,
           cMemory := "SS2_A4_32DO_DO_Vars".DO27.cMemory,
           iCounterIn := "SS2_A4_32DO_DO_Vars".DO27.iCounterIn,
           iCounterOut := "SS2_A4_32DO_DO_Vars".DO27.iCounterOut,
           xOutput => "SS2_A4_32DO_DO_Vars".DO27.xOutput);
   "DO12.04.27" := "SS2_A4_32DO_DO_Vars".DO27.xOutput;
END_REGION

REGION Network 28: DQd3
   RUNG wire#powerrail
      "DOvar"(iFuncSystem := "SS2_A4_32DO_DO_Vars".DO28.iFuncSystemID, iFuncVar := "SS2_A4_32DO_DO_Vars".DO28.iFuncVar, xOutput => "SS2_A4_32DO_DO_Vars".DO28.xInput)
   END_RUNG
   RUNG wire#powerrail
      "DOadv"(xInput := "SS2_A4_32DO_DO_Vars".DO28.xInput, xInversion := "SS2_A4_32DO_DO_Vars".DO28.xInversion, cMOA := "SS2_A4_32DO_DO_Vars".DO28.cMOA, xMemoryOut := "SS2_A4_32DO_DO_Vars".DO28.xMemoryOut, xMemoryIn := "SS2_A4_32DO_DO_Vars".DO28.xMemoryIn, cMemory := "SS2_A4_32DO_DO_Vars".DO28.cMemory, iCounterIn := "SS2_A4_32DO_DO_Vars".DO28.iCounterIn, iCounterOut := "SS2_A4_32DO_DO_Vars".DO28.iCounterOut, xOutput => "SS2_A4_32DO_DO_Vars".DO28.xOutput)
   END_RUNG
   RUNG wire#powerrail
      Contact( "SS2_A4_32DO_DO_Vars".DO28.xOutput )
      Coil( "DO12.04.28" )
   END_RUNG
   // the same network as SCL:
   "DOvar"(iFuncSystem := "SS2_A4_32DO_DO_Vars".DO28.iFuncSystemID,
           iFuncVar := "SS2_A4_32DO_DO_Vars".DO28.iFuncVar,
           xOutput => "SS2_A4_32DO_DO_Vars".DO28.xInput);
   "DOadv"(xInput := "SS2_A4_32DO_DO_Vars".DO28.xInput,
           xInversion := "SS2_A4_32DO_DO_Vars".DO28.xInversion,
           cMOA := "SS2_A4_32DO_DO_Vars".DO28.cMOA,
           xMemoryOut := "SS2_A4_32DO_DO_Vars".DO28.xMemoryOut,
           xMemoryIn := "SS2_A4_32DO_DO_Vars".DO28.xMemoryIn,
           cMemory := "SS2_A4_32DO_DO_Vars".DO28.cMemory,
           iCounterIn := "SS2_A4_32DO_DO_Vars".DO28.iCounterIn,
           iCounterOut := "SS2_A4_32DO_DO_Vars".DO28.iCounterOut,
           xOutput => "SS2_A4_32DO_DO_Vars".DO28.xOutput);
   "DO12.04.28" := "SS2_A4_32DO_DO_Vars".DO28.xOutput;
END_REGION

REGION Network 29: DQd4
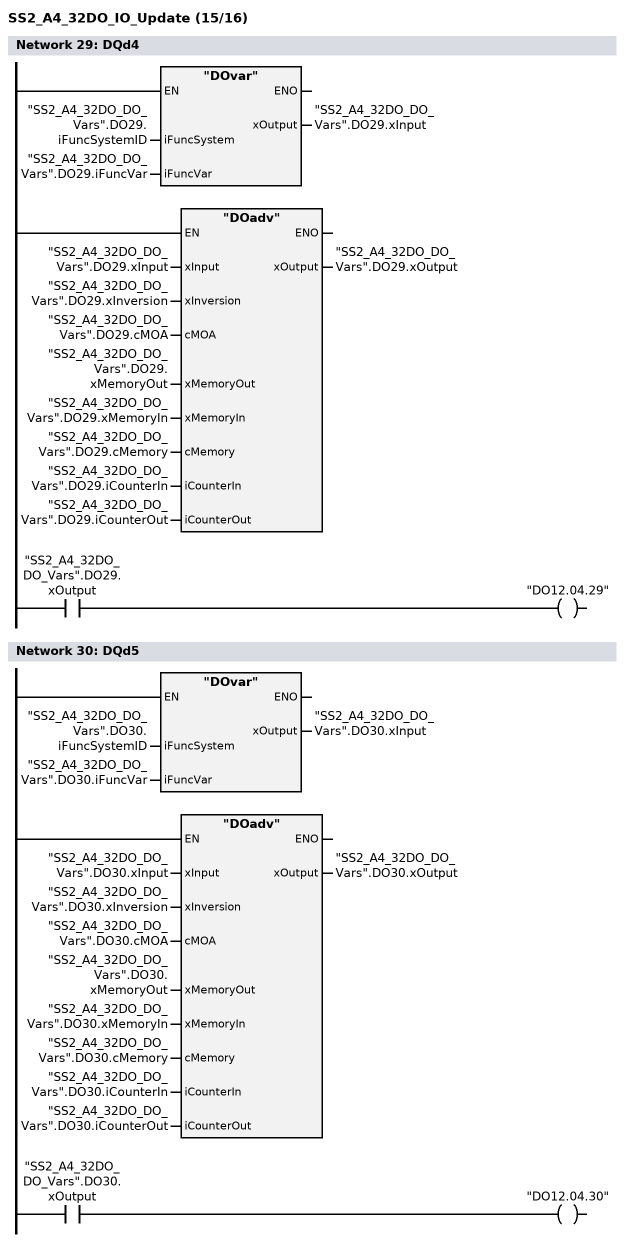
   RUNG wire#powerrail
      "DOvar"(iFuncSystem := "SS2_A4_32DO_DO_Vars".DO29.iFuncSystemID, iFuncVar := "SS2_A4_32DO_DO_Vars".DO29.iFuncVar, xOutput => "SS2_A4_32DO_DO_Vars".DO29.xInput)
   END_RUNG
   RUNG wire#powerrail
      "DOadv"(xInput := "SS2_A4_32DO_DO_Vars".DO29.xInput, xInversion := "SS2_A4_32DO_DO_Vars".DO29.xInversion, cMOA := "SS2_A4_32DO_DO_Vars".DO29.cMOA, xMemoryOut := "SS2_A4_32DO_DO_Vars".DO29.xMemoryOut, xMemoryIn := "SS2_A4_32DO_DO_Vars".DO29.xMemoryIn, cMemory := "SS2_A4_32DO_DO_Vars".DO29.cMemory, iCounterIn := "SS2_A4_32DO_DO_Vars".DO29.iCounterIn, iCounterOut := "SS2_A4_32DO_DO_Vars".DO29.iCounterOut, xOutput => "SS2_A4_32DO_DO_Vars".DO29.xOutput)
   END_RUNG
   RUNG wire#powerrail
      Contact( "SS2_A4_32DO_DO_Vars".DO29.xOutput )
      Coil( "DO12.04.29" )
   END_RUNG
   // the same network as SCL:
   "DOvar"(iFuncSystem := "SS2_A4_32DO_DO_Vars".DO29.iFuncSystemID,
           iFuncVar := "SS2_A4_32DO_DO_Vars".DO29.iFuncVar,
           xOutput => "SS2_A4_32DO_DO_Vars".DO29.xInput);
   "DOadv"(xInput := "SS2_A4_32DO_DO_Vars".DO29.xInput,
           xInversion := "SS2_A4_32DO_DO_Vars".DO29.xInversion,
           cMOA := "SS2_A4_32DO_DO_Vars".DO29.cMOA,
           xMemoryOut := "SS2_A4_32DO_DO_Vars".DO29.xMemoryOut,
           xMemoryIn := "SS2_A4_32DO_DO_Vars".DO29.xMemoryIn,
           cMemory := "SS2_A4_32DO_DO_Vars".DO29.cMemory,
           iCounterIn := "SS2_A4_32DO_DO_Vars".DO29.iCounterIn,
           iCounterOut := "SS2_A4_32DO_DO_Vars".DO29.iCounterOut,
           xOutput => "SS2_A4_32DO_DO_Vars".DO29.xOutput);
   "DO12.04.29" := "SS2_A4_32DO_DO_Vars".DO29.xOutput;
END_REGION

REGION Network 30: DQd5
   RUNG wire#powerrail
      "DOvar"(iFuncSystem := "SS2_A4_32DO_DO_Vars".DO30.iFuncSystemID, iFuncVar := "SS2_A4_32DO_DO_Vars".DO30.iFuncVar, xOutput => "SS2_A4_32DO_DO_Vars".DO30.xInput)
   END_RUNG
   RUNG wire#powerrail
      "DOadv"(xInput := "SS2_A4_32DO_DO_Vars".DO30.xInput, xInversion := "SS2_A4_32DO_DO_Vars".DO30.xInversion, cMOA := "SS2_A4_32DO_DO_Vars".DO30.cMOA, xMemoryOut := "SS2_A4_32DO_DO_Vars".DO30.xMemoryOut, xMemoryIn := "SS2_A4_32DO_DO_Vars".DO30.xMemoryIn, cMemory := "SS2_A4_32DO_DO_Vars".DO30.cMemory, iCounterIn := "SS2_A4_32DO_DO_Vars".DO30.iCounterIn, iCounterOut := "SS2_A4_32DO_DO_Vars".DO30.iCounterOut, xOutput => "SS2_A4_32DO_DO_Vars".DO30.xOutput)
   END_RUNG
   RUNG wire#powerrail
      Contact( "SS2_A4_32DO_DO_Vars".DO30.xOutput )
      Coil( "DO12.04.30" )
   END_RUNG
   // the same network as SCL:
   "DOvar"(iFuncSystem := "SS2_A4_32DO_DO_Vars".DO30.iFuncSystemID,
           iFuncVar := "SS2_A4_32DO_DO_Vars".DO30.iFuncVar,
           xOutput => "SS2_A4_32DO_DO_Vars".DO30.xInput);
   "DOadv"(xInput := "SS2_A4_32DO_DO_Vars".DO30.xInput,
           xInversion := "SS2_A4_32DO_DO_Vars".DO30.xInversion,
           cMOA := "SS2_A4_32DO_DO_Vars".DO30.cMOA,
           xMemoryOut := "SS2_A4_32DO_DO_Vars".DO30.xMemoryOut,
           xMemoryIn := "SS2_A4_32DO_DO_Vars".DO30.xMemoryIn,
           cMemory := "SS2_A4_32DO_DO_Vars".DO30.cMemory,
           iCounterIn := "SS2_A4_32DO_DO_Vars".DO30.iCounterIn,
           iCounterOut := "SS2_A4_32DO_DO_Vars".DO30.iCounterOut,
           xOutput => "SS2_A4_32DO_DO_Vars".DO30.xOutput);
   "DO12.04.30" := "SS2_A4_32DO_DO_Vars".DO30.xOutput;
END_REGION

REGION Network 31: DQd6
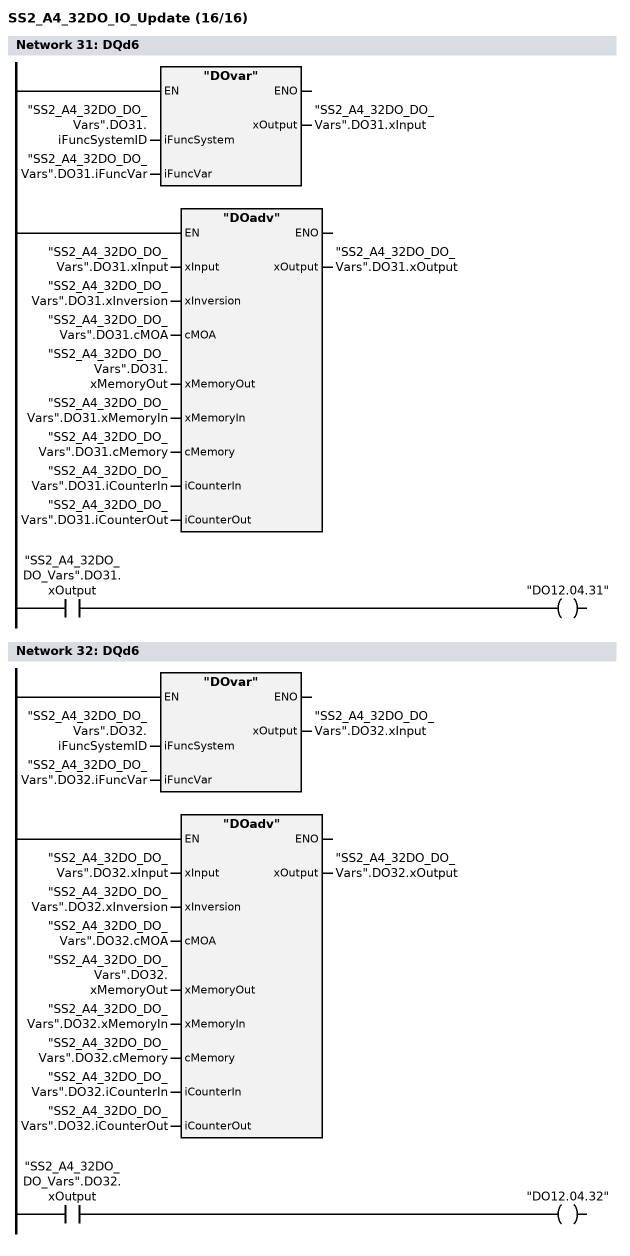
   RUNG wire#powerrail
      "DOvar"(iFuncSystem := "SS2_A4_32DO_DO_Vars".DO31.iFuncSystemID, iFuncVar := "SS2_A4_32DO_DO_Vars".DO31.iFuncVar, xOutput => "SS2_A4_32DO_DO_Vars".DO31.xInput)
   END_RUNG
   RUNG wire#powerrail
      "DOadv"(xInput := "SS2_A4_32DO_DO_Vars".DO31.xInput, xInversion := "SS2_A4_32DO_DO_Vars".DO31.xInversion, cMOA := "SS2_A4_32DO_DO_Vars".DO31.cMOA, xMemoryOut := "SS2_A4_32DO_DO_Vars".DO31.xMemoryOut, xMemoryIn := "SS2_A4_32DO_DO_Vars".DO31.xMemoryIn, cMemory := "SS2_A4_32DO_DO_Vars".DO31.cMemory, iCounterIn := "SS2_A4_32DO_DO_Vars".DO31.iCounterIn, iCounterOut := "SS2_A4_32DO_DO_Vars".DO31.iCounterOut, xOutput => "SS2_A4_32DO_DO_Vars".DO31.xOutput)
   END_RUNG
   RUNG wire#powerrail
      Contact( "SS2_A4_32DO_DO_Vars".DO31.xOutput )
      Coil( "DO12.04.31" )
   END_RUNG
   // the same network as SCL:
   "DOvar"(iFuncSystem := "SS2_A4_32DO_DO_Vars".DO31.iFuncSystemID,
           iFuncVar := "SS2_A4_32DO_DO_Vars".DO31.iFuncVar,
           xOutput => "SS2_A4_32DO_DO_Vars".DO31.xInput);
   "DOadv"(xInput := "SS2_A4_32DO_DO_Vars".DO31.xInput,
           xInversion := "SS2_A4_32DO_DO_Vars".DO31.xInversion,
           cMOA := "SS2_A4_32DO_DO_Vars".DO31.cMOA,
           xMemoryOut := "SS2_A4_32DO_DO_Vars".DO31.xMemoryOut,
           xMemoryIn := "SS2_A4_32DO_DO_Vars".DO31.xMemoryIn,
           cMemory := "SS2_A4_32DO_DO_Vars".DO31.cMemory,
           iCounterIn := "SS2_A4_32DO_DO_Vars".DO31.iCounterIn,
           iCounterOut := "SS2_A4_32DO_DO_Vars".DO31.iCounterOut,
           xOutput => "SS2_A4_32DO_DO_Vars".DO31.xOutput);
   "DO12.04.31" := "SS2_A4_32DO_DO_Vars".DO31.xOutput;
END_REGION

REGION Network 32: DQd6
   RUNG wire#powerrail
      "DOvar"(iFuncSystem := "SS2_A4_32DO_DO_Vars".DO32.iFuncSystemID, iFuncVar := "SS2_A4_32DO_DO_Vars".DO32.iFuncVar, xOutput => "SS2_A4_32DO_DO_Vars".DO32.xInput)
   END_RUNG
   RUNG wire#powerrail
      "DOadv"(xInput := "SS2_A4_32DO_DO_Vars".DO32.xInput, xInversion := "SS2_A4_32DO_DO_Vars".DO32.xInversion, cMOA := "SS2_A4_32DO_DO_Vars".DO32.cMOA, xMemoryOut := "SS2_A4_32DO_DO_Vars".DO32.xMemoryOut, xMemoryIn := "SS2_A4_32DO_DO_Vars".DO32.xMemoryIn, cMemory := "SS2_A4_32DO_DO_Vars".DO32.cMemory, iCounterIn := "SS2_A4_32DO_DO_Vars".DO32.iCounterIn, iCounterOut := "SS2_A4_32DO_DO_Vars".DO32.iCounterOut, xOutput => "SS2_A4_32DO_DO_Vars".DO32.xOutput)
   END_RUNG
   RUNG wire#powerrail
      Contact( "SS2_A4_32DO_DO_Vars".DO32.xOutput )
      Coil( "DO12.04.32" )
   END_RUNG
   // the same network as SCL:
   "DOvar"(iFuncSystem := "SS2_A4_32DO_DO_Vars".DO32.iFuncSystemID,
           iFuncVar := "SS2_A4_32DO_DO_Vars".DO32.iFuncVar,
           xOutput => "SS2_A4_32DO_DO_Vars".DO32.xInput);
   "DOadv"(xInput := "SS2_A4_32DO_DO_Vars".DO32.xInput,
           xInversion := "SS2_A4_32DO_DO_Vars".DO32.xInversion,
           cMOA := "SS2_A4_32DO_DO_Vars".DO32.cMOA,
           xMemoryOut := "SS2_A4_32DO_DO_Vars".DO32.xMemoryOut,
           xMemoryIn := "SS2_A4_32DO_DO_Vars".DO32.xMemoryIn,
           cMemory := "SS2_A4_32DO_DO_Vars".DO32.cMemory,
           iCounterIn := "SS2_A4_32DO_DO_Vars".DO32.iCounterIn,
           iCounterOut := "SS2_A4_32DO_DO_Vars".DO32.iCounterOut,
           xOutput => "SS2_A4_32DO_DO_Vars".DO32.xOutput);
   "DO12.04.32" := "SS2_A4_32DO_DO_Vars".DO32.xOutput;
END_REGION
END_FUNCTION
